       #FB_STATE_TCP_RECONNECTING:
         REGION FB_STATE_TCP_RECONNECTING
           IF #tempTsendcStatus = #TSENDC_EST_OK THEN
             #statErrorAutoCleared := FALSE;
             // Update edge detection
             #statPublishOld := #tempPublish;
             #statSubscribeOld := #tempSubscribe;
             #statUnsubscribeOld := #tempUnsubscribe;
             //Monitor Connection
             #statFBState := #FB_STATE_OPERATING_MONITOR_TCP;
             // Begin MQTT Connection
             #statMqttConnectState := #MQTT_CONNECT_STATE_BUILD_PAKET;
           END_IF;
         END_REGION FB_STATE_TCP_RECONNECTING
       #FB_STATE_DISABLING: // Disabling active
         REGION DISABLING FB
           //  Disabling, e.g. closing connections, etc.
           // When disabling is complete the bit #statDisablingCompleted must be set
           // When MQTT is connected, send disconnect
           IF #statMqttConnectState = #MQTT_CONNECT_STATE_CONNECTED THEN
             IF #statTsendcReq = TRUE THEN
               //Interrupt any existing send jobs
               #statTsendcReq := FALSE;
             ELSE
               // INIT
               #statSendBufferPos := 0;
               //Build fixed Header
               //Message Type
               #statSendBuffer[#statSendBufferPos] := #MQTT_MSG_TYPE_DISCONNECT;
               #statSendBufferPos += 1;
               //Remaining Length (must be O)
               #statSendBuffer[#statSendBufferPos] := #REMAINIG_LEN_0;
               #statSendBufferPos += 1;
               //send request
               #statTsendcLen := #statSendBufferPos;
               #statTsendcReq := TRUE;
               #statMqttConnectState := #MQTT_CONNECT_STATE_DISCONNECTED;
             END_IF;
           ELSE
             //Disable TCP Connection
             #statTsendcReq := FALSE;
             #statTsendcEnable := FALSE;
             #statEnableTimerCommandWatchdog := TRUE;
           END_IF;
           // When TCP connection is closed
           IF #tempTsendcStatus = #TSENDC_DISCONNECTED THEN
             #statEnableTimerCommandWatchdog := FALSE;
             #statDisablingCompleted := TRUE;
           ELSIF #instTimerCommandWatchdog.Q THEN
             #statEnableTimerCommandWatchdog := FALSE;
             #statDisablingCompleted := TRUE;
           END_IF;
         END_REGION DISABLING FB
       ELSE // Undefined state in state machine reached
         #statStatus := #ERR_UNDEFINED_STATE;
         #statErrorUserCleared := TRUE;
     END_CASE;
   END_REGION STATE_MACHINE

   REGION OUTPUTS
     // Write outputs
     IF (#statDisablingCompleted = TRUE) THEN
       // Reset outputs if disabling completed
       #statValid := FALSE;
       #statBusy := FALSE;
       #statError := FALSE;
       #statDone := FALSE;
       #statErrorUserCleared := FALSE;
       #statErrorAutoCleared := FALSE;
       #statStatus := #STATUS_NO_CALL;
       // Reset application specific outputs
       #statRcvMsgStatus := #MSG_DECODE_STATUS_NO_NEW_MSG;
       #statRcvMsgDataLen := 0;

     ELSIF (#statErrorUserCleared = TRUE) AND (#statError = FALSE) THEN
       // Error can only be cleared by user; rising edge at enable input is needed to continue 
       #statValid := FALSE;
       #statBusy := FALSE;
       #statDone := FALSE;
       #statError := TRUE;
       // Write diagnostics
       #diagnostics.status := #statStatus;
       #diagnostics.subfunctionStatus := #statSubfunctionStatus;
       #diagnostics.stateNumber := #statFBErrorState;
       // execution aborted --> set state no processing
       #statTsendcEnable := FALSE; // Terminate Connection, no reason keep it up.
       #statFBState := #FB_STATE_NO_PROCESSING;
       #statMqttConnectState := #MQTT_CONNECT_STATE_NO_PROCESSING;
       #statMqttCommandState := #MQTT_COMMAND_STATE_NO_PROCESSING;
       #statRcvMsgDecodeState := #MSG_DECODE_STATE_NO_PROCESSING;

     ELSIF (#statErrorAutoCleared = TRUE) AND (#statError = FALSE) THEN
       // Error can be reset by FB automatically
       #statValid := FALSE;
       #statBusy := TRUE;
       #statError := TRUE;
       #statDone := FALSE;

       // Write diagnostics
       #diagnostics.status := #statStatus;
       #diagnostics.subfunctionStatus := #statSubfunctionStatus;
       #diagnostics.stateNumber := #statFBErrorState;
       // Handling of autocleared error
       CASE #statStatus OF
           //Just signal error and reset autocleared error afterwards.
         #ERR_MQTT_PAKET_ID_INVALID, #ERR_MQTT_SUBACK_FAILURE, #ERR_MQTT_CONNECT_TIMEOUT,
         #ERR_MQTT_COMMAND_SEND_TIMEOUT, #ERR_MQTT_COMMAND_MULTIPLE_INPUT, #ERR_CNT_EXCEEDS_ARRAY_DIMENSION,
         #ERR_MQTT_COMMAND_PUBLISH_TOPIC_INVALID, #ERR_QOS_INVALID, #ERR_MQTT_COMMAND_SUBSCRIBE_TOPIC_INVALID:
           #statErrorAutoCleared := FALSE;

         ELSE  // Statement section ELSE
           ;
       END_CASE;

     ELSIF (#statErrorAutoCleared = FALSE) AND (#statErrorUserCleared = FALSE) AND (#statError = TRUE) THEN
       // If autocleared error is acknowledged
       #statValid := TRUE;
       #statBusy := TRUE;
       #statError := FALSE;
       #statDone := FALSE;

       //   this line  more detailed status information is used instead of "#STATUS_SUBSEQUENT_CALL"
       CASE #statStatus OF
         #ERR_TCP_RECONNECTING, #ERR_MQTT_CONNECT_TIMEOUT:  // Reconnecting ok, start Mqtt reconnnect
           //set status
           #statStatus := #STATUS_MQTT_CONNECTING;
           //in the following status codes status stays connected. 
         #ERR_MQTT_PAKET_ID_INVALID, #ERR_MQTT_SUBACK_FAILURE, #ERR_MQTT_COMMAND_SEND_TIMEOUT,
         #ERR_MQTT_COMMAND_MULTIPLE_INPUT, #ERR_CNT_EXCEEDS_ARRAY_DIMENSION, #ERR_MQTT_COMMAND_PUBLISH_TOPIC_INVALID,
         #ERR_QOS_INVALID, #ERR_MQTT_COMMAND_SUBSCRIBE_TOPIC_INVALID:
           #statStatus := #STATUS_MQTT_CONNECTED;
         ELSE  // Statement section ELSE
           ;
       END_CASE;
     END_IF;

     // Write static values to outputs
     #valid := #statValid;
     #busy := #statBusy;
     #error := #statError;
     #status := #statStatus;
     //block sets ENO automatically:
     //ENO := TRUE;
     //Write application specific static values to outputs
     #done := #statDone;
     #receivedMsgStatus := #statRcvMsgStatus;
     #receivedMsgDataLen := #statRcvMsgDataLen;
   END_REGION OUTPUTS
END_FUNCTION_BLOCK

FUNCTION "TransmitMqttData" : Void   // FC17, SCL
{ S7_Optimized_Access := 'TRUE' }
VERSION : 0.1
BEGIN
END_FUNCTION

// folder: LMQTT/Utilities

FUNCTION "LMQTT_ConvertToUtf8" : Void   // FC15, SCL
TITLE = LMQTT_ConvertToUtf8
{ S7_Optimized_Access := 'TRUE' }
AUTHOR : SIEMENS
FAMILY : LMQTT
VERSION : 1.0
// Function to convert a WCHAR to a UTF-8 conformant byte sequence
   VAR_INPUT
      character : WChar;   // Character that shall be converted to UTF-8
   END_VAR
   VAR_OUTPUT
      convertedUtf8 : DWord;   // UTF-8 conformant byte sequence. B0 stores first Byte, B1 second and B2 third Byte. B3 is not used
      bytesUsed : USInt;   // Amount of Bytes converted. Ranges from 1 to 3.
      error : Bool;   // TRUE: An error occurred during the execution of the FC
      status : Word;   // 16#0000 - 16#7FFF: Status of the FC, 16#8000 - 16#FFFF: Error identification
   END_VAR
   VAR_TEMP
      tempStatus : Word;   // temp value for output 'status'
      tempConvertedUtf8 : DWord;   // temp value for output 'convertedUtf8'
      tempBytesUsed : USInt;   // temp value for output 'bytesUsed'
      tempCharacter : WChar;   // temp value for input 'character'
   END_VAR
   // Ret_Val : No return for this FC - see error and status output
   VAR CONSTANT
      STATUS_NO_ERROR : Word := 16#0000;   // no error status
      STATUS_EXECUTION_FINISHED : Word := 16#0000;   // Execution finished without errors
      ERR_UNDEFINED : Word := 16#8000;   // Error due to an undefined case
      USINT_NULL : USInt := 0;   // Init value with 0
      DWORD_NULL : DWord := 16#0000_0000;   // Init value with 0
      EMPTY_WCHAR : WChar := WCHAR#' ';   // Empty WChar for comparison
      BELOW_7F : Word := 16#007F;   // Upper limit for character if only one Byte used
      BELOW_7FF : Word := 16#07FF;   // Upper limit for character if two Byte used
      BELOW_MAX_FFFF : Word := 16#FFFF;   // Upper limit for character if three Byte used
      BYTE_3F : Byte := 16#3F;   // Conversion Value
      BYTE_80 : Byte := 16#80;   // Conversion Value
      BYTE_C0 : Byte := 16#C0;   // Conversion Value
      BYTE_E0 : Byte := 16#E0;   // Conversion Value
      USINT_ONE : USInt := 1;   // Const Value to assign amount of bytes used
      USINT_TWO : USInt := 2;   // Const Value to assign amount of bytes used
      USINT_THREE : USInt := 3;   // Const Value to assign amount of bytes used
   END_VAR
BEGIN
   REGION BLOCK INFO HEADER
       //=============================================================================
       // SIEMENS AG
       // (c)Copyright 2020
       //-----------------------------------------------------------------------------
       // Library:       LMQTT
       // Tested with:   CPU 1516-3 PN/DP V2.8
       // Engineering:   TIA Portal V16
       // Restrictions:  --
       // Requirements:  --
       // Functionality: Converts a single WChar Character to a valid UTF-8 encoded byte sequence and saves this to a DWord.
       //                The amount of bytes saved is stored in bytesUsed Output.
       //-----------------------------------------------------------------------------
       // Change log table:
       // Version    Date         Expert in charge         Changes applied
       // 03.00.00   01.10.2020   Siemens Online Support   First released version
       //=============================================================================
   END_REGION

   REGION INITIALISATION  
       // Initialize functionality: reset of variables, diagnostics, etc.
       #tempConvertedUtf8 := #DWORD_NULL;
       #tempBytesUsed := #USINT_NULL;
       #tempStatus := #STATUS_NO_ERROR;
       //assign temp value from input:
        #tempCharacter := #character;

   END_REGION

   REGION PROGRAM LOGIC
       // Use this region for application specific code
       IF #tempCharacter = #EMPTY_WCHAR THEN
           //will be only 1 byte occupied
           #tempConvertedUtf8 := WCHAR_TO_DWORD(#tempCharacter);
           #tempBytesUsed := #USINT_ONE;
       ELSIF (WCHAR_TO_WORD(#tempCharacter) <= (#BELOW_7F)) THEN
           //will be only 1 byte occupied
           #tempConvertedUtf8 := WCHAR_TO_DWORD(#tempCharacter);
           #tempBytesUsed := #USINT_ONE;
       ELSIF (WCHAR_TO_WORD(#tempCharacter) <= (#BELOW_7FF)) THEN
           //will be 2 byte occupied
           #tempConvertedUtf8.%B1 := (WCHAR_TO_BYTE(#tempCharacter) AND #BYTE_3F) OR #BYTE_80;
           #tempConvertedUtf8.%B0 := WORD_TO_BYTE(SHR(IN := WCHAR_TO_WORD(#tempCharacter), N := 6)) OR #BYTE_C0;
           #tempBytesUsed := #USINT_TWO;
       ELSIF (WCHAR_TO_WORD(#tempCharacter) <= (#BELOW_MAX_FFFF)) THEN
           //will be 3 byte occupied
           #tempConvertedUtf8.%B2 := (WCHAR_TO_BYTE(#tempCharacter) AND #BYTE_3F) OR #BYTE_80;
           #tempConvertedUtf8.%B1 := (WORD_TO_BYTE(SHR(IN := WCHAR_TO_WORD(#tempCharacter), N := 6)) AND #BYTE_3F) OR #BYTE_80;
           #tempConvertedUtf8.%B0 := WORD_TO_BYTE(SHR(IN := WCHAR_TO_WORD(#tempCharacter), N := 12)) OR #BYTE_E0;
           #tempBytesUsed := #USINT_THREE;
       END_IF;
   END_REGION

   REGION OUTPUTS
       // Write application specific temp values to outputs
       #bytesUsed := #tempBytesUsed;
       #convertedUtf8 := #tempConvertedUtf8;
       // Write error and status
       #error := #tempStatus.%X15;
       #status := #tempStatus;
       // ENO mechanism is not used --> ENO := TRUE;
       ENO := TRUE;
   END_REGION
END_FUNCTION

// folder: LossManagement

FUNCTION "CopyLoss" : Void   // FC12, SCL
{ S7_Optimized_Access := 'TRUE' }
VERSION : 0.1
   VAR_INPUT
      In : "MachineEventDatatype";
   END_VAR
   VAR_OUTPUT
      Out : "MachineEventListView";
   END_VAR
BEGIN
   #Out."no." := #In.id;
   #Out.LossCode := #In.losscode;
   //#Out.assign_losscode := #In.assign_losscode;
   #Out.Description := "SettingsDB_LossDescription".loss_descriptions[#In.losscode].description;//#In.description;
   //#Out.StartTime:= #In.StartTime;
   //#Out.StartTimeAsStr:= #In.StartTimeAsStr;
   //#Out.EndTime:= #In.EndTime;

   "DTL_to_String"("DTL" := #In.startTime,
                   OutputStr => #Out.StartDateAsStr);


   "DTL_to_String"("DTL" := #In.endTime,
                   OutputStr => #Out.EndDateAsStr);

   "TimeToString"(timeValue := UDINT_TO_TIME(#In.duration),
                  OutputStr => #Out.DurationAsStr);
   //#Out.EndTimeAsStr:= #In.EndTimeAsStr;
   //#Out.DurationAsStr:= #In.DurationAsStr;
   //#Out.Duration := #In.Duration;
   #Out.StatusServer := #In.statusServer;
END_FUNCTION

FUNCTION "CheckDiffLoss" : Void   // FC13, SCL
{ S7_Optimized_Access := 'TRUE' }
VERSION : 0.1
   VAR_INPUT
      "IN 1" : "MachineEventDatatype";
      "IN 2" : "MachineEventListView";
   END_VAR
   VAR_OUTPUT
      IsDiff : Bool;
   END_VAR
BEGIN
   #IsDiff := #"IN 1".id <> #"IN 2"."no.";
   #IsDiff := #IsDiff OR (#"IN 1".losscode <> #"IN 2".LossCode);

   //#IsDiff := #IsDiff OR (#"IN 1".description <> #"IN 2".description);
   // #IsDiff := #IsDiff OR (#"IN 1".StartTimeAsStr <> #"IN 2".StartTimeAsStr);
   // #IsDiff := #IsDiff OR (#"IN 1".EndTimeAsStr <> #"IN 2".EndTimeAsStr);
   // #IsDiff := #IsDiff OR (#"IN 1".DurationAsStr <> #"IN 2".DurationAsStr);
   #IsDiff := #IsDiff OR (#"IN 1".statusServer <> #"IN 2".StatusServer);
END_FUNCTION

FUNCTION "ListviewDisplayLoss" : Void   // FC14, SCL
{ S7_Optimized_Access := 'TRUE' }
VERSION : 0.1
   VAR_INPUT
      MinSlotId : Int;
      MaxSlotId : Int;
   END_VAR
   VAR_TEMP
      tmpIsDiff : Bool;
   END_VAR
BEGIN
   // FOR "bufferLossId" := 1 TO 30 DO
   //     IF "BuffersLoss_DB".buffer_loss_in_shift["bufferLossId"].id > 0 THEN

   //         IF ("slotId" > #MinSlotId) AND ("slotId" <= #MaxSlotId) THEN
   //             IF "listviewId" <= 10 THEN

   //                 // "CheckDiffLoss"("IN 1" := "BuffersLoss_DB".buffer_loss_in_shift["bufferLossId"],
   //                 //                 "IN 2" := "DB_Machine".machine_event_listview["listviewId"],
   //                 //                 IsDiff => #tmpIsDiff);
   //                 #tmpIsDiff := TRUE;
   //                 IF #tmpIsDiff THEN
   //                     "CopyLoss"(In := "BuffersLoss_DB".buffer_loss_in_shift["bufferLossId"],
   //                                Out => "DB_Machine".machine_event_listview["listviewId"]);
   //                 END_IF;
   //                 //
   //                 "DB_Machine".machine_event_listview["listviewId"].IsHaveData := TRUE;
   //                 "listviewId" := "listviewId" + 1;
   //             END_IF;
   //             //
   //         END_IF;

   //         "slotId" := "slotId" + 1;
   //     END_IF;
   // END_FOR;
END_FUNCTION

FUNCTION "ShowDescriptionLossByGroupId" : Void   // FC22, SCL
{ S7_Optimized_Access := 'TRUE' }
VERSION : 0.1
   VAR_INPUT
      GroupId : USInt;
      PageCurrent : UDInt;
      NumberDataEachPage : USInt;
   END_VAR
   VAR_OUTPUT
      ListDescriptionResult : Array[1..10] of String[30];
   END_VAR
   VAR_TEMP
      IndexFor : USInt;
      ListDescriptionResultTemp : Array[1..100] of String[30];
      IndexLossResult : USInt;
   END_VAR
BEGIN
   IF #GroupId>=1 AND #GroupId<=10 THEN
       #IndexLossResult := 1;
       FOR #IndexFor := 1 TO 100 DO
           IF "SettingsDB_LossDescription".loss_descriptions[#IndexFor].group_id = #GroupId THEN // Statement section FOR
               #ListDescriptionResultTemp[#IndexLossResult] := "SettingsDB_LossDescription".loss_descriptions[#IndexFor].description;
               #IndexLossResult += 1;
           END_IF;
       END_FOR;

       FOR #IndexFor := 1 TO 10 DO
           IF #IndexLossResult <= 10 THEN
               #ListDescriptionResult[#IndexLossResult] := '';
               //#ListDescriptionResult[#IndexLossResult].group_id := 0;
               #IndexLossResult += 1;
           ELSE
               EXIT;
           END_IF;
       END_FOR;

   ELSIF #GroupId=0 THEN //Case All
       FOR #IndexFor := 1 TO 10 DO
           #ListDescriptionResult[#IndexFor] := "SettingsDB_LossDescription".loss_descriptions[#IndexFor + (#PageCurrent - 1) * #NumberDataEachPage].description;
       END_FOR;
   END_IF;
END_FUNCTION

FUNCTION "MappingLossGroup" : Void   // FC23, SCL
{ S7_Optimized_Access := 'TRUE' }
VERSION : 0.1
   VAR_TEMP
      indexFor : USInt;
   END_VAR
BEGIN
   FOR #indexFor := 1 TO 10 DO
       IF "SettingsDB_LossDescription".loss_name_group[#indexFor] = '' THEN
           "DB_DataHMI".VisibleCheckboxLossGroup[#indexFor] := FALSE;
       ELSE
           "DB_DataHMI".VisibleCheckboxLossGroup[#indexFor] := TRUE;
       END_IF;

       "DB_DataHMI".LossGroupHmiDTO[#indexFor] := "SettingsDB_LossDescription".loss_name_group[#indexFor];
   END_FOR;
END_FUNCTION

FUNCTION "GetBufferHistoricalShowHMI" : Void   // FC24, SCL
{ S7_Optimized_Access := 'TRUE' }
VERSION : 0.1
   VAR_INPUT
      page_current_hmi : UDInt;
   END_VAR
   VAR_TEMP
      index_for : USInt;
      index_buffer : UDInt;
      page_hmi_cvt : UDInt;
   END_VAR
BEGIN
   IF #page_current_hmi>=1 THEN
       #page_hmi_cvt := #page_current_hmi MOD 10;
       IF #page_hmi_cvt=0 THEN
           #page_hmi_cvt := 10;
       END_IF;

       #index_buffer := (#page_hmi_cvt - 1) * 5;

       FOR #index_for:= 1 TO 5 DO
           IF "BuffersLoss_DB".buffer_loss_in_historical[#index_buffer + #index_for].id > 0 THEN
               "DB_DataHMI".DataLossHistoricalShowHmiDTO[#index_for]."no." := UDINT_TO_UINT((#page_current_hmi - 1) * 5 + #index_for);
               "DB_DataHMI".DataLossHistoricalShowHmiDTO[#index_for].LossCode := "BuffersLoss_DB".buffer_loss_in_historical[#index_buffer + #index_for].losscode;

               "Cvt_Duration_to_String"("Time(ms)" := "BuffersLoss_DB".buffer_loss_in_historical[#index_buffer + #index_for].duration,
                                        ConvertTimeToStr => "DB_DataHMI".DataLossHistoricalShowHmiDTO[#index_for].DurationAsStr);

               "DTL_to_DateString"("DTL" := "BuffersLoss_DB".buffer_loss_in_historical[#index_buffer + #index_for].startTime,
                                   DateTimeString => "DB_DataHMI".DataLossHistoricalShowHmiDTO[#index_for].StartDateAsStr);
               "DTL_to_TimeString"("DTL" := "BuffersLoss_DB".buffer_loss_in_historical[#index_buffer + #index_for].startTime,
                                   DateTimeString => "DB_DataHMI".DataLossHistoricalShowHmiDTO[#index_for].StartTimeAsStr);

               "DTL_to_DateString"("DTL" := "BuffersLoss_DB".buffer_loss_in_historical[#index_buffer + #index_for].endTime,
                                   DateTimeString => "DB_DataHMI".DataLossHistoricalShowHmiDTO[#index_for].EndDateAsStr);
               "DTL_to_TimeString"("DTL" := "BuffersLoss_DB".buffer_loss_in_historical[#index_buffer + #index_for].endTime,
                                   DateTimeString => "DB_DataHMI".DataLossHistoricalShowHmiDTO[#index_for].EndTimeAsStr);

               IF  "DB_DataHMI".DataLossHistoricalShowHmiDTO[#index_for].LossCode>0 AND  "DB_DataHMI".DataLossHistoricalShowHmiDTO[#index_for].LossCode<=100 THEN
                   "DB_DataHMI".DataLossHistoricalShowHmiDTO[#index_for].Description := "SettingsDB_LossDescription".loss_descriptions["DB_DataHMI".DataLossHistoricalShowHmiDTO[#index_for].LossCode].description;
                   IF "SettingsDB_LossDescription".loss_descriptions["DB_DataHMI".DataLossHistoricalShowHmiDTO[#index_for].LossCode].group_id>0 AND
                       "SettingsDB_LossDescription".loss_descriptions["DB_DataHMI".DataLossHistoricalShowHmiDTO[#index_for].LossCode].group_id<=10 THEN
                       "DB_DataHMI".DataLossHistoricalShowHmiDTO[#index_for].GroupLossReason := "SettingsDB_LossDescription".loss_name_group["SettingsDB_LossDescription".loss_descriptions["DB_DataHMI".DataLossHistoricalShowHmiDTO[#index_for].LossCode].group_id];
                   END_IF;
               END_IF;

               "DB_DataHMI".DataLossHistoricalShowHmiDTO[#index_for].IsHaveData := TRUE;
           END_IF;
       END_FOR;
   END_IF;
END_FUNCTION

FUNCTION "LogStartLoss" : Void   // FC26, SCL
{ S7_Optimized_Access := 'TRUE' }
VERSION : 0.1
BEGIN
   "GLobalDB_LossManagementDB".current_status_machine.startTime := "GlobalDB_RTC".RTC_Local;
END_FUNCTION

FUNCTION "LogEndLoss" : Void   // FC27, SCL
{ S7_Optimized_Access := 'TRUE' }
VERSION : 0.1
BEGIN
   "GLobalDB_LossManagementDB".current_status_machine.startTime := "GlobalDB_RTC".RTC_Local;
END_FUNCTION

FUNCTION "CheckMoveDataLossCurrent" : Void   // FC28, SCL
{ S7_Optimized_Access := 'TRUE' }
VERSION : 0.1
BEGIN
   "GLobalDB_LossManagementDB".current_status_machine.endTime := "GlobalDB_RTC".RTC_Local;
   "GLobalDB_LossManagementDB".current_status_machine.duration := "GLobalDB_LossManagementDB"."duration_status_curent(ms)";
   "GLobalDB_LossManagementDB".current_status_machine.id := "GLobalDB_LossManagementDB".id_loss;


   "DTL_to_StringV2"("DTL":="GLobalDB_LossManagementDB".current_status_machine.startTime,
                     DateTimeString=>"DB_DataHMI".PageHomeStartTimeStatusCurrent);

   "DTL_to_StringV2"("DTL" := "GLobalDB_LossManagementDB".current_status_machine.endTime,
                     DateTimeString => "DB_DataHMI".PageHomeEndTimeStatusCurrent);

   "Cvt_Duration_to_String"("Time(ms)":="GLobalDB_LossManagementDB".current_status_machine.duration,
                            ConvertTimeToStr=>"DB_DataHMI".PageHomeDurationStatusCurrent);


   //Kiểm tra Loss hiện tại quá tgian cài đặt sẽ bắt buộc "AssignLoss"
   IF ("GLobalDB_LossManagementDB".current_status_machine.duration/1000) >= ("DataSetting"."TimeThresholdShowWarningAssignLoss(s)")
       AND "DB_DataHMI".FlagCancelAssignLossCurrent=FALSE
       AND ("DB_DataHMI".MachineStatus=2 OR "DB_DataHMI".MachineStatus=3) THEN
       "DB_DataHMI".PageHomeBitShowAssignLoss := TRUE;
       "DB_DataHMI".TypeAssignLoss := 3;
   ELSE
       "DB_DataHMI".PageHomeBitShowAssignLoss := FALSE;
   END_IF;


   //Kiểm tra  AssignLoss hiện tại để move data
   IF "DB_DataHMI".EventAssignLossCurrent=TRUE THEN
       "DB_DataHMI".StartTimeAssignLossCurrent := "DB_DataHMI".PageHomeStartTimeStatusCurrent;
       "DB_DataHMI".EndTimeAssignLossCurrent := "DB_DataHMI".PageHomeEndTimeStatusCurrent;
       "DB_DataHMI".DurationAssignLossCurrent := "DB_DataHMI".PageHomeDurationStatusCurrent;
   END_IF;


   //MOve tamj ddons khacsh
   IF "DB_DataHMI".MachineStatus=2 OR "DB_DataHMI".MachineStatus=3 THEN
       "GLobalDB_LossManagementDB".current_status_machine.statusServer := UINT_TO_USINT("DB_DataHMI".MachineStatus);

       "BuffersLoss_DB".buffer_loss_in_shift["GLobalDB_LossManagementDB".index_buffer_loss_in_shift_current].startTime := "GLobalDB_LossManagementDB".current_status_machine.startTime;
       "BuffersLoss_DB".buffer_loss_in_shift["GLobalDB_LossManagementDB".index_buffer_loss_in_shift_current].endTime := "GlobalDB_RTC".RTC_Defaul;
       "BuffersLoss_DB".buffer_loss_in_shift["GLobalDB_LossManagementDB".index_buffer_loss_in_shift_current].id := "GLobalDB_LossManagementDB".current_status_machine.id;
       "BuffersLoss_DB".buffer_loss_in_shift["GLobalDB_LossManagementDB".index_buffer_loss_in_shift_current].duration := "GLobalDB_LossManagementDB".current_status_machine.duration;
       "BuffersLoss_DB".buffer_loss_in_shift["GLobalDB_LossManagementDB".index_buffer_loss_in_shift_current].statusServer := "GLobalDB_LossManagementDB".current_status_machine.statusServer;
   END_IF;
END_FUNCTION

FUNCTION "LogLoss" : Void   // FC33, SCL
{ S7_Optimized_Access := 'TRUE' }
VERSION : 0.1
   VAR_INPUT
      status : UInt;   // 1: Runnig, 2Stop, 3Idle
   END_VAR
   VAR_IN_OUT
      index_buffer : USInt;   // 1=>100
   END_VAR
BEGIN
   IF #index_buffer>=1 AND #index_buffer<=100 THEN
       "BuffersLoss_DB".buffer_loss_in_shift[#index_buffer] := "GLobalDB_LossManagementDB".current_status_machine;
       "BuffersLoss_DB".buffer_loss_in_shift[#index_buffer].statusServer := UINT_TO_USINT(#status);

       "GLobalDB_LossManagementDB".id_loss += 1;
       //"DB_Machine".NumberLossInShift += 1;
       #index_buffer += 1;
       IF #index_buffer > 100 THEN
           #index_buffer := 1;
       END_IF;
   ELSE
       #index_buffer := 1;
   END_IF;
END_FUNCTION

FUNCTION "CheckIndexRowAssignLoss" : Void   // FC42, SCL
{ S7_Optimized_Access := 'TRUE' }
VERSION : 0.1
   VAR_TEMP
      index_for : USInt;
      group_id : UInt;
   END_VAR
BEGIN
   FOR #index_for := 1 TO 5 DO
       IF "DB_DataHMI".EventIndexRowInShift[#index_for]=TRUE THEN
           "DB_DataHMI".IndexRowAssignLoss := #index_for;
           "DB_DataHMI".EventIndexRowInShift[#index_for] := FALSE;

           "DB_DataHMI".TypeAssignLoss := 1;
       END_IF;
   END_FOR;

   FOR #index_for := 1 TO 5 DO
       IF "DB_DataHMI".EventIndexRowHistorical[#index_for] = TRUE THEN
           "DB_DataHMI".IndexRowAssignLoss := #index_for;
           "DB_DataHMI".EventIndexRowHistorical[#index_for] := FALSE;

           "DB_DataHMI".TypeAssignLoss := 2;
       END_IF;
   END_FOR;



   IF "DB_DataHMI".TypeAssignLoss=1 THEN //LOss In Shift
       "DB_DataHMI".LossReasonSelectId := 0;
       IF "DB_DataHMI".IndexRowAssignLoss>=1 AND "DB_DataHMI".IndexRowAssignLoss<=5 THEN
           "DB_DataHMI".StartTimeAssignLossCurrent := CONCAT(IN1 := "DB_DataHMI".DataLossInShiftShowHmiDTO["DB_DataHMI".IndexRowAssignLoss].StartDateAsStr,
                                                             IN2 := ' ',
                                                             IN3 := "DB_DataHMI".DataLossInShiftShowHmiDTO["DB_DataHMI".IndexRowAssignLoss].StartTimeAsStr);

           "DB_DataHMI".EndTimeAssignLossCurrent := CONCAT(IN1 := "DB_DataHMI".DataLossInShiftShowHmiDTO["DB_DataHMI".IndexRowAssignLoss].EndDateAsStr,
                                                             IN2 := ' ',
                                                             IN3 := "DB_DataHMI".DataLossInShiftShowHmiDTO["DB_DataHMI".IndexRowAssignLoss].EndTimeAsStr);
           "DB_DataHMI".DurationAssignLossCurrent := "DB_DataHMI".DataLossInShiftShowHmiDTO["DB_DataHMI".IndexRowAssignLoss].DurationAsStr;

           //Tim thông tin AssignLoss của Loss hiện tại nếu có
           "ResetCheckBoxLossReason"();
           IF "DB_DataHMI".DataLossInShiftShowHmiDTO["DB_DataHMI".IndexRowAssignLoss].LossCode>0 AND "DB_DataHMI".DataLossInShiftShowHmiDTO["DB_DataHMI".IndexRowAssignLoss].LossCode<=10 THEN
               "DB_DataHMI".CheckboxLossReason["DB_DataHMI".DataLossInShiftShowHmiDTO["DB_DataHMI".IndexRowAssignLoss].LossCode] := 1;

               "DB_DataHMI".LossReasonSelectId := "DB_DataHMI".DataLossInShiftShowHmiDTO["DB_DataHMI".IndexRowAssignLoss].LossCode;

               "ResetCheckBoxLossGroup"();
               #group_id := "SettingsDB_LossDescription".loss_descriptions["DB_DataHMI".DataLossInShiftShowHmiDTO["DB_DataHMI".IndexRowAssignLoss].LossCode].group_id;
               IF #group_id>0 AND #group_id<=10 THEN
                   "DB_DataHMI".CheckboxLossGroup[#group_id] := 1;
               END_IF;

           END_IF;
       END_IF;
       "DB_DataHMI".TypeAssignLoss := 0;
   ELSIF "DB_DataHMI".TypeAssignLoss=2 THEN //Historical
       "DB_DataHMI".LossReasonSelectId := 0;
       IF "DB_DataHMI".IndexRowAssignLoss >= 1 AND "DB_DataHMI".IndexRowAssignLoss <= 5 THEN
           "DB_DataHMI".StartTimeAssignLossCurrent := CONCAT(IN1 := "DB_DataHMI".DataLossHistoricalShowHmiDTO["DB_DataHMI".IndexRowAssignLoss].StartDateAsStr,
                                                             IN2 := ' ',
                                                             IN3 := "DB_DataHMI".DataLossHistoricalShowHmiDTO["DB_DataHMI".IndexRowAssignLoss].EndTimeAsStr);

           "DB_DataHMI".EndTimeAssignLossCurrent := CONCAT(IN1 := "DB_DataHMI".DataLossHistoricalShowHmiDTO["DB_DataHMI".IndexRowAssignLoss].EndDateAsStr,
                                                           IN2 := ' ',
                                                           IN3 := "DB_DataHMI".DataLossHistoricalShowHmiDTO["DB_DataHMI".IndexRowAssignLoss].EndTimeAsStr);
           "DB_DataHMI".DurationAssignLossCurrent := "DB_DataHMI".DataLossHistoricalShowHmiDTO["DB_DataHMI".IndexRowAssignLoss].DurationAsStr;


           //Tim thông tin AssignLoss của Loss hiện tại nếu có
           "ResetCheckBoxLossReason"();
           IF "DB_DataHMI".DataLossHistoricalShowHmiDTO["DB_DataHMI".IndexRowAssignLoss].LossCode > 0 AND
               "DB_DataHMI".DataLossHistoricalShowHmiDTO["DB_DataHMI".IndexRowAssignLoss].LossCode <= 10 THEN
               "DB_DataHMI".CheckboxLossReason["DB_DataHMI".DataLossHistoricalShowHmiDTO["DB_DataHMI".IndexRowAssignLoss].LossCode] := 1;

               "DB_DataHMI".LossReasonSelectId := "DB_DataHMI".DataLossHistoricalShowHmiDTO["DB_DataHMI".IndexRowAssignLoss].LossCode;

               "ResetCheckBoxLossGroup"();
               #group_id := "SettingsDB_LossDescription".loss_descriptions["DB_DataHMI".DataLossHistoricalShowHmiDTO["DB_DataHMI".IndexRowAssignLoss].LossCode].group_id;
               IF #group_id > 0 AND #group_id <= 10 THEN
                   "DB_DataHMI".CheckboxLossGroup[#group_id] := 1;
               END_IF;

           END_IF;
       END_IF;
       "DB_DataHMI".TypeAssignLoss := 0;
   ELSIF "DB_DataHMI".TypeAssignLoss=3 THEN //Loss Current
       "DB_DataHMI".StartTimeAssignLossCurrent := "DB_DataHMI".PageHomeStartTimeStatusCurrent;
       "DB_DataHMI".EndTimeAssignLossCurrent := "DB_DataHMI".PageHomeEndTimeStatusCurrent;
       "DB_DataHMI".DurationAssignLossCurrent := "DB_DataHMI".PageHomeDurationStatusCurrent;
   END_IF;


   //Kiểm tra Action Cancel nếu người ta bỏ qua AssignLoss hiện tại
   IF "DB_DataHMI".FlagCancelAssignLossCurrent = TRUE AND "DB_DataHMI".TypeAssignLoss=3 THEN
       "DB_DataHMI".PageHomeBitShowAssignLoss := FALSE;
   END_IF;
END_FUNCTION

FUNCTION "FindSyncLossInShift" : Void   // FC63, SCL
{ S7_Optimized_Access := 'TRUE' }
VERSION : 0.1
   VAR_TEMP
      index_for : USInt;
      compare_start_time : Bool;
      compare_end_time : Bool;
   END_VAR
BEGIN
   FOR #index_for := 1 TO 100 DO
       "CompareDTL"(DTL_Input1:="DB_Server".LossInShiftAssign.startTime,
                                          DTL_Input2:="BuffersLoss_DB".buffer_loss_in_shift[#index_for].startTime,
                                          Result=>#compare_start_time);

                             "CompareDTL"(DTL_Input1 := "DB_Server".LossInShiftAssign.endTime,
                                           DTL_Input2 := "BuffersLoss_DB".buffer_loss_in_shift[#index_for].endTime,
                                           Result => #compare_end_time);

      IF #compare_start_time = TRUE AND #compare_end_time = TRUE THEN
          "BuffersLoss_DB".buffer_loss_in_shift[#index_for].losscode := "DB_Server".LossInShiftAssign.losscode;
          EXIT;
      END_IF;
   END_FOR;
END_FUNCTION

FUNCTION "ResStatusSearchLossHistorical" : Void   // FC69, SCL
{ S7_Optimized_Access := 'TRUE' }
VERSION : 0.1
   VAR_IN_OUT
      value_flag : UInt;
   END_VAR
BEGIN
   IF #value_flag=2 THEN
       "DB_DataHMI".EventBitShowPopupLoading := FALSE;
       IF "DB_Server".PageHistorical.TotalData=0 THEN
           "DB_DataHMI".EventBitShowNoDataHistorical := TRUE;
           "DB_Server".ActionSearchLossHistorical := 3;
       END_IF;
   ELSIF #value_flag=4 THEN
       "DB_DataHMI".EventBitShowPopupLoading := FALSE;
       "DB_DataHMI".EventBitShowPopupErrorFormatDaySearch := TRUE;
       #value_flag := 3;
   END_IF;
END_FUNCTION

// folder: RTC

FUNCTION "RTC" : Void   // FC6, LAD
{ S7_Optimized_Access := 'TRUE' }
VERSION : 0.1
   VAR_OUTPUT
      Year : UInt;
      Month : UInt;
      Day : UInt;
      Hour : UInt;
      Minute : UInt;
      Second : UInt;
   END_VAR
   VAR_TEMP
      max : USInt;
      min : USInt;
   END_VAR
BEGIN

REGION Network 1
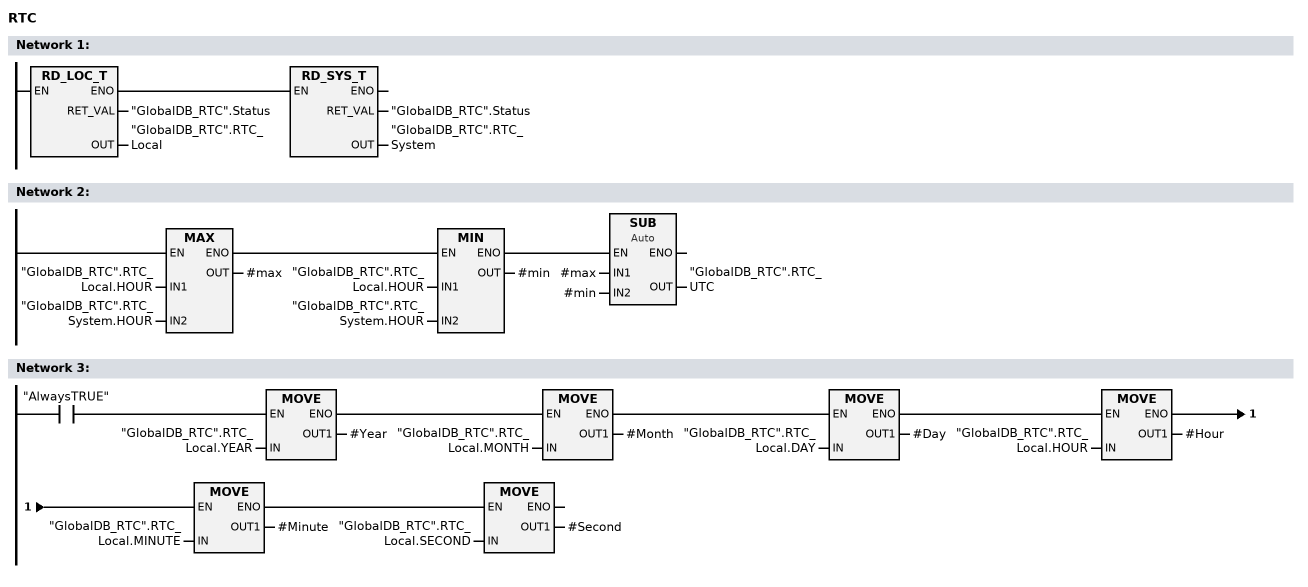
   // ENO of a box is taken as its EN; it also drops when the box reports an error
   "GlobalDB_RTC".Status := RD_LOC_T(OUT => "GlobalDB_RTC".RTC_Local);
   "GlobalDB_RTC".Status := RD_SYS_T(OUT => "GlobalDB_RTC".RTC_System);
END_REGION

REGION Network 2
   #max := MAX(IN1 := "GlobalDB_RTC".RTC_Local.HOUR, IN2 := "GlobalDB_RTC".RTC_System.HOUR);
   #min := MIN(IN1 := "GlobalDB_RTC".RTC_Local.HOUR, IN2 := "GlobalDB_RTC".RTC_System.HOUR);
   "GlobalDB_RTC".RTC_UTC := #max - #min;
END_REGION

REGION Network 3
   RUNG wire#powerrail
      Contact( "AlwaysTRUE" )
      Move(in := "GlobalDB_RTC".RTC_Local.YEAR, out1 => #Year)
      Move(in := "GlobalDB_RTC".RTC_Local.MONTH, out1 => #Month)
      Move(in := "GlobalDB_RTC".RTC_Local.DAY, out1 => #Day)
      Move(in := "GlobalDB_RTC".RTC_Local.HOUR, out1 => #Hour)
      Move(in := "GlobalDB_RTC".RTC_Local.MINUTE, out1 => #Minute)
      Move(in := "GlobalDB_RTC".RTC_Local.SECOND, out1 => #Second)
   END_RUNG
   // the same network as SCL:
   IF "AlwaysTRUE" THEN
       #Year := "GlobalDB_RTC".RTC_Local.YEAR;
       #Month := "GlobalDB_RTC".RTC_Local.MONTH;
       #Day := "GlobalDB_RTC".RTC_Local.DAY;
       #Hour := "GlobalDB_RTC".RTC_Local.HOUR;
       #Minute := "GlobalDB_RTC".RTC_Local.MINUTE;
       #Second := "GlobalDB_RTC".RTC_Local.SECOND;
   END_IF;
END_REGION
END_FUNCTION

FUNCTION "SyncTimeFromPC" : Void   // FC66, LAD
{ S7_Optimized_Access := 'TRUE' }
VERSION : 0.1
   VAR_IN_OUT
      EventSync : Bool;
   END_VAR
BEGIN

REGION Network 1: Set và Get lại thời gian PLC khi có sự kiện update
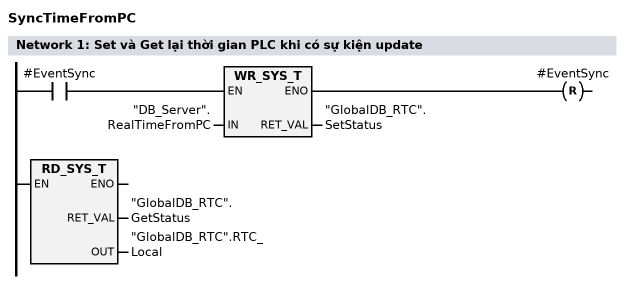
   // ENO of a box is taken as its EN; it also drops when the box reports an error
   IF #EventSync THEN
       "GlobalDB_RTC".SetStatus := WR_SYS_T(IN := "DB_Server".RealTimeFromPC);
       #EventSync := FALSE;
   END_IF;
   "GlobalDB_RTC".GetStatus := RD_SYS_T(OUT => "GlobalDB_RTC".RTC_Local);
END_REGION
END_FUNCTION

// folder: Sensor-Counter

FUNCTION_BLOCK "CounterFB"   // FB3, LAD
{ S7_Optimized_Access := 'TRUE' }
VERSION : 0.1
   VAR_INPUT
      bCounterTrigger : Bool;
      bResetCounter : Bool;
      TonFilter_x1ms : UInt := 10;   // ms
      ToffFilter_x1ms : UInt := 10;   // ms
   END_VAR
   VAR_IN_OUT
      CounterOut : UDInt;
   END_VAR
   VAR RETAIN
      P_tmp : Bool;
      N_tmp : Bool;
   END_VAR
   VAR
      Ton_start : Bool;
      Toff_start : Bool;
   END_VAR
   VAR RETAIN
      IEC_Ton : IEC_TIMER;
      IEC_Toff : IEC_TIMER;
      bTmp : Bool;
   END_VAR
   VAR
      Ton_x1ms : Time;
      Toff_x1ms : Time;
   END_VAR
   VAR_TEMP   // added for the SCL form of the ladder/FBD networks
      _w1 : Bool;
   END_VAR
BEGIN

REGION Network 1
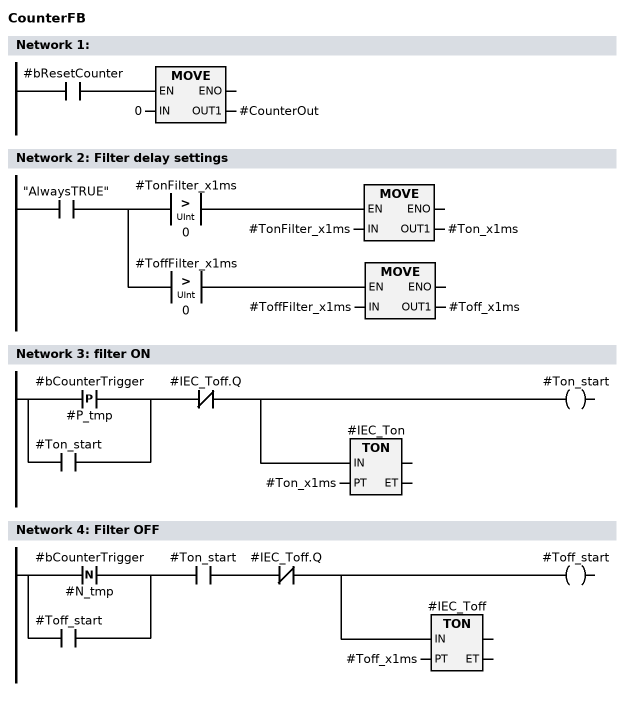
   RUNG wire#powerrail
      Contact( #bResetCounter )
      Move(in := 0, out1 => #CounterOut)
   END_RUNG
   // the same network as SCL:
   IF #bResetCounter THEN #CounterOut := 0; END_IF;
END_REGION

REGION Network 2: Filter delay settings
   RUNG wire#powerrail
      Contact( "AlwaysTRUE" )
      wire#w1
      { S7_Templates := "SrcType := UInt" } GT_Contact(in1 := #TonFilter_x1ms, in2 := 0)
      Move(in := #TonFilter_x1ms, out1 => #Ton_x1ms)
   END_RUNG
   RUNG wire#w1
      { S7_Templates := "SrcType := UInt" } GT_Contact(in1 := #ToffFilter_x1ms, in2 := 0)
      Move(in := #ToffFilter_x1ms, out1 => #Toff_x1ms)
   END_RUNG
   // the same network as SCL:
   IF "AlwaysTRUE" AND (#TonFilter_x1ms > 0) THEN #Ton_x1ms := #TonFilter_x1ms; END_IF;
   IF "AlwaysTRUE" AND (#ToffFilter_x1ms > 0) THEN #Toff_x1ms := #ToffFilter_x1ms; END_IF;
END_REGION

REGION Network 3: filter ON
   #_w1 := #bCounterTrigger AND NOT #P_tmp;   // rising edge of #bCounterTrigger
   #P_tmp := #bCounterTrigger;
   #Ton_start := (#_w1 OR #Ton_start) AND NOT #IEC_Toff.Q;
   #IEC_Ton.TON(IN := #Ton_start, PT := #Ton_x1ms);
END_REGION

REGION Network 4: Filter OFF
   #_w1 := NOT #bCounterTrigger AND #N_tmp;   // falling edge of #bCounterTrigger
   #N_tmp := #bCounterTrigger;
   #Toff_start := (#_w1 OR #Toff_start) AND #Ton_start AND NOT #IEC_Toff.Q;
   #IEC_Toff.TON(IN := #Toff_start, PT := #Toff_x1ms);
END_REGION

REGION Network 5 (SCL)
   IF #Ton_start AND NOT #bTmp THEN
       #CounterOut := #CounterOut + 1;
   END_IF;
   #bTmp := #Ton_start;
END_REGION
END_FUNCTION_BLOCK

// folder: Sensor-Speed

FUNCTION_BLOCK "1.2 Speed_Sensor"   // FB1, LAD
{ S7_Optimized_Access := 'TRUE' }
VERSION : 0.1
   VAR_INPUT
      "InputTimeSpeed(time_each_pulse)" : Time;
      NumberOfGears : UInt;
      Index : Int;
   END_VAR
   VAR_OUTPUT
      "OutputSpeed(rpm)" : DInt;
      "TimePerPulse(x1ms)" : DInt;
   END_VAR
   VAR RETAIN
      bThroudoutStart : Bool;
      TimeSpeed : Time;
      speed_tmp : Array[1..3] of DInt;
      speed_tmpidx : Int;
      previous_speed_tmpidx : Int;
      CurrentSpeed : DInt;
   END_VAR
   VAR
      real_tmp : Real;
      real_tmp_1 : Real;
      dint_tmp : DInt;
      real_tmp_2 : Real;
      number_of_gears_tmp : Real;
   END_VAR
   VAR_TEMP   // added for the SCL form of the ladder/FBD networks
      _w1 : Bool;
   END_VAR
BEGIN

REGION Network 1
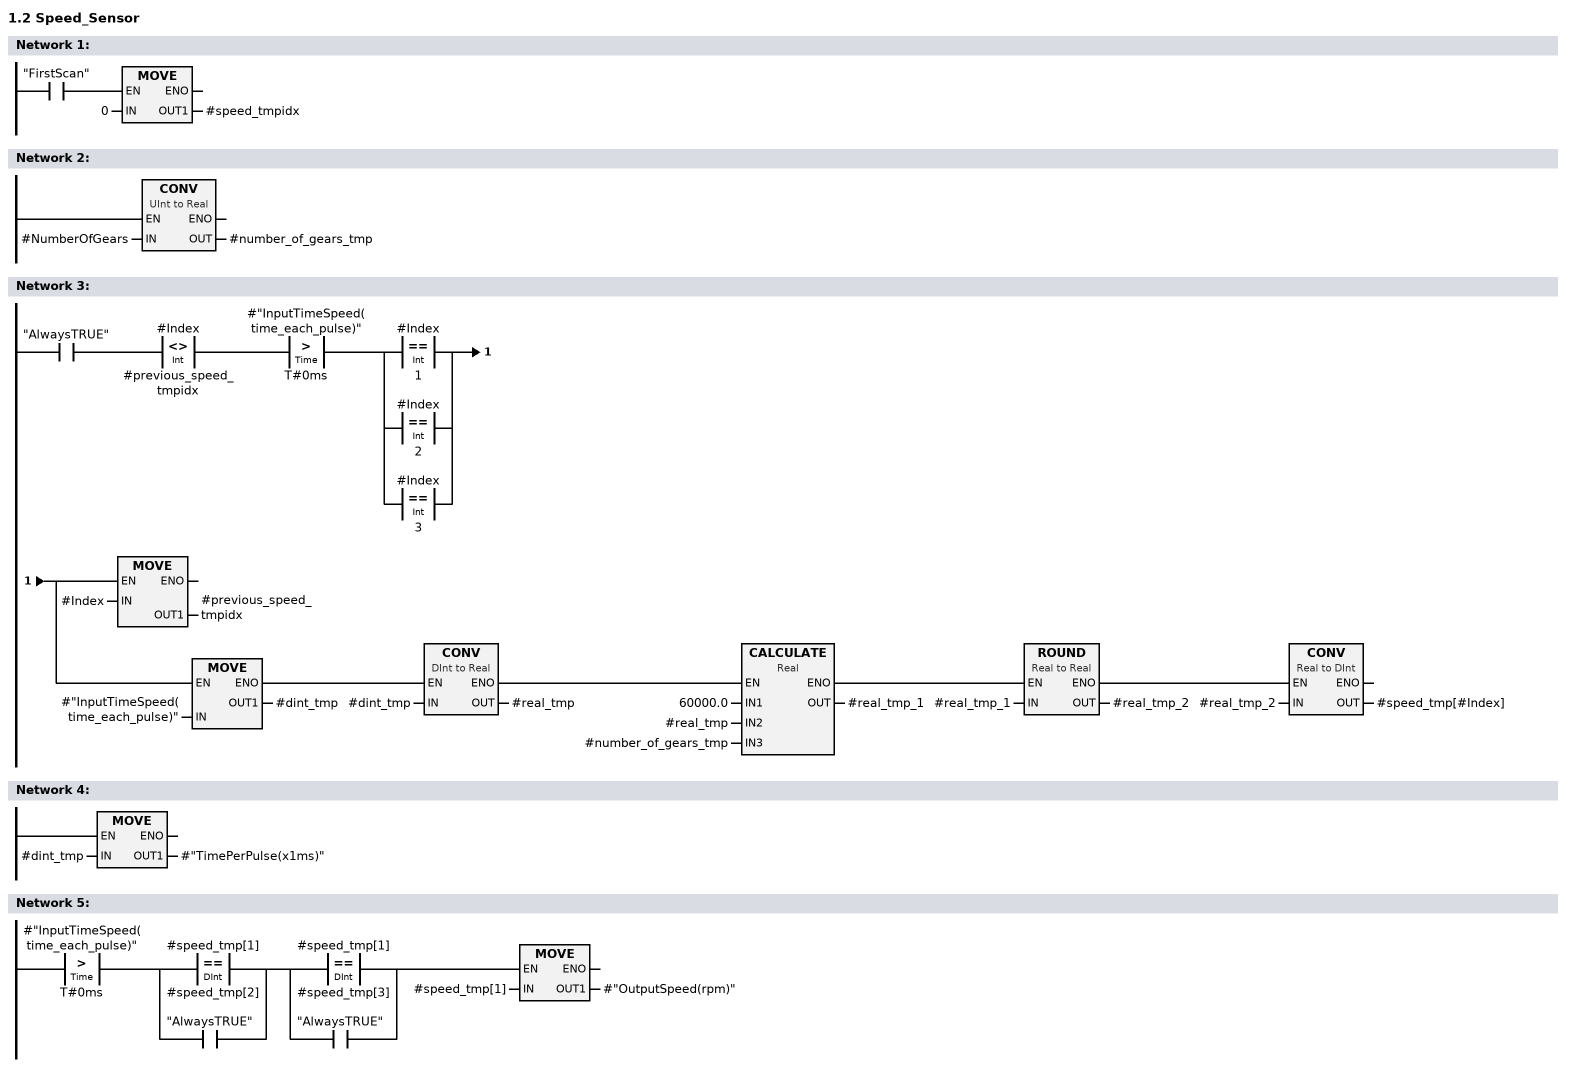
   RUNG wire#powerrail
      Contact( "FirstScan" )
      Move(in := 0, out1 => #speed_tmpidx)
   END_RUNG
   // the same network as SCL:
   IF "FirstScan" THEN #speed_tmpidx := 0; END_IF;
END_REGION

REGION Network 2
   RUNG wire#powerrail
      { S7_Templates := "[SrcType := UInt, DestType := Real]" } Convert(in := #NumberOfGears, out => #number_of_gears_tmp)
   END_RUNG
   // the same network as SCL:
   #number_of_gears_tmp := UINT_TO_REAL(#NumberOfGears);
END_REGION

REGION Network 3
   RUNG wire#powerrail
      Contact( "AlwaysTRUE" )
      { S7_Templates := "SrcType := Int" } NE_Contact(in1 := #Index, in2 := #previous_speed_tmpidx)
      { S7_Templates := "SrcType := Time" } GT_Contact(in1 := #"InputTimeSpeed(time_each_pulse)", in2 := T#0ms)
      wire#w1
      { S7_Templates := "SrcType := Int" } EQ_Contact(in1 := #Index, in2 := 1)
      wire#w2
      Move(in := #Index, out1 => #previous_speed_tmpidx)
   END_RUNG
   RUNG wire#w1
      { S7_Templates := "SrcType := Int" } EQ_Contact(in1 := #Index, in2 := 2)
   END_RUNG wire#w2
   RUNG wire#w1
      { S7_Templates := "SrcType := Int" } EQ_Contact(in1 := #Index, in2 := 3)
   END_RUNG wire#w2
   RUNG wire#w2
      Move(in := #"InputTimeSpeed(time_each_pulse)", out1 => #dint_tmp)
      { S7_Templates := "[SrcType := DInt, DestType := Real]" } Convert(in := #dint_tmp, out => #real_tmp)
      { S7_Templates := "SrcType := Real"; S7_Expression := "IN1/(IN2*IN3)" } Calculate(in1 := 60000.0, in2 := #real_tmp, in3 := #number_of_gears_tmp, out => #real_tmp_1)
      { S7_Templates := "[SrcType := Real, DestType := Real]" } Round(in := #real_tmp_1, out => #real_tmp_2)
      { S7_Templates := "[SrcType := Real, DestType := DInt]" } Convert(in := #real_tmp_2, out => #speed_tmp[#Index])
   END_RUNG
   // the same network as SCL:
   #_w1 := "AlwaysTRUE" AND (#Index <> #previous_speed_tmpidx) AND (#"InputTimeSpeed(time_each_pulse)" > T#0ms) AND ((#Index = 1) OR (#Index = 2) OR (#Index = 3));
   IF #_w1 THEN
       #previous_speed_tmpidx := #Index;
       #dint_tmp := #"InputTimeSpeed(time_each_pulse)";
       #real_tmp := DINT_TO_REAL(#dint_tmp);
       #real_tmp_1 := 60000.0/(#real_tmp*#number_of_gears_tmp);
       #real_tmp_2 := ROUND(#real_tmp_1);
       #speed_tmp[#Index] := REAL_TO_DINT(#real_tmp_2);
   END_IF;
END_REGION

REGION Network 4
   RUNG wire#powerrail
      Move(in := #dint_tmp, out1 => #"TimePerPulse(x1ms)")
   END_RUNG
   // the same network as SCL:
   #"TimePerPulse(x1ms)" := #dint_tmp;
END_REGION

REGION Network 5
   RUNG wire#powerrail
      { S7_Templates := "SrcType := Time" } GT_Contact(in1 := #"InputTimeSpeed(time_each_pulse)", in2 := T#0ms)
      wire#w1
      { S7_Templates := "SrcType := DInt" } EQ_Contact(in1 := #speed_tmp[1], in2 := #speed_tmp[2])
      wire#w2
      { S7_Templates := "SrcType := DInt" } EQ_Contact(in1 := #speed_tmp[1], in2 := #speed_tmp[3])
      wire#w3
      Move(in := #speed_tmp[1], out1 => #"OutputSpeed(rpm)")
   END_RUNG
   RUNG wire#w1
      Contact( "AlwaysTRUE" )
   END_RUNG wire#w2
   RUNG wire#w2
      Contact( "AlwaysTRUE" )
   END_RUNG wire#w3
   // the same network as SCL:
   IF (#"InputTimeSpeed(time_each_pulse)" > T#0ms) AND ((#speed_tmp[1] = #speed_tmp[2]) OR "AlwaysTRUE") AND ((#speed_tmp[1] = #speed_tmp[3]) OR "AlwaysTRUE") THEN
       #"OutputSpeed(rpm)" := #speed_tmp[1];
   END_IF;
END_REGION
END_FUNCTION_BLOCK

FUNCTION_BLOCK "1.3 Speed Interrupt"   // FB2, LAD
{ S7_Optimized_Access := 'TRUE' }
VERSION : 0.1
   VAR_OUTPUT
      TimeSpeed : Time;
      speed_tmpidx : Int;
   END_VAR
   VAR RETAIN
      ".IEC_TIMER_SensorSpeed" : IEC_TIMER;
      bSpeedStart : Bool;
   END_VAR
BEGIN

REGION Network 1
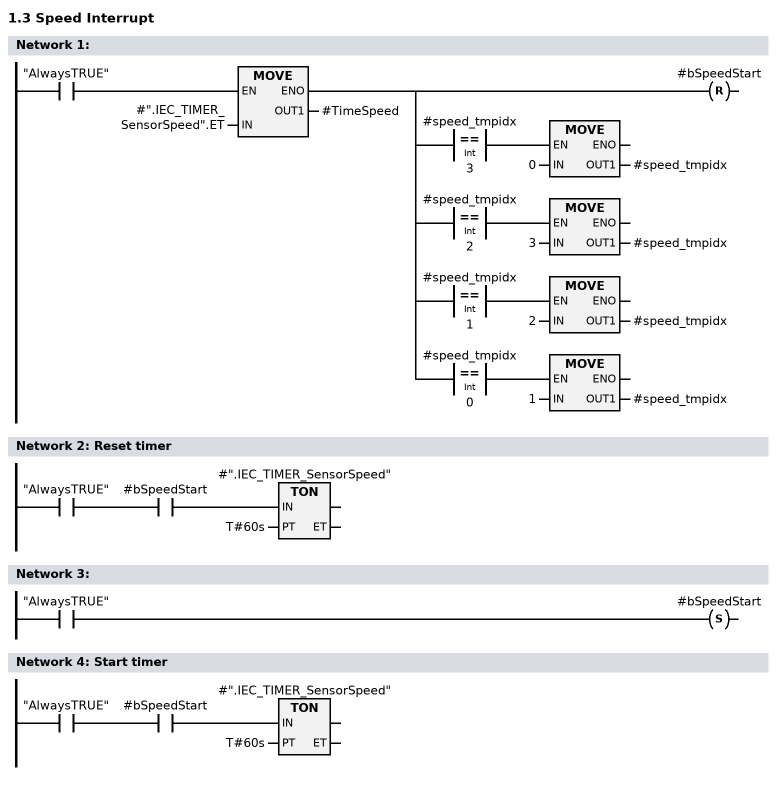
   RUNG wire#powerrail
      Contact( "AlwaysTRUE" )
      Move(in := #".IEC_TIMER_SensorSpeed".ET, out1 => #TimeSpeed)
      wire#w1
      R_Coil( #bSpeedStart )
   END_RUNG
   RUNG wire#w1
      { S7_Templates := "SrcType := Int" } EQ_Contact(in1 := #speed_tmpidx, in2 := 3)
      Move(in := 0, out1 => #speed_tmpidx)
   END_RUNG
   RUNG wire#w1
      { S7_Templates := "SrcType := Int" } EQ_Contact(in1 := #speed_tmpidx, in2 := 2)
      Move(in := 3, out1 => #speed_tmpidx)
   END_RUNG
   RUNG wire#w1
      { S7_Templates := "SrcType := Int" } EQ_Contact(in1 := #speed_tmpidx, in2 := 1)
      Move(in := 2, out1 => #speed_tmpidx)
   END_RUNG
   RUNG wire#w1
      { S7_Templates := "SrcType := Int" } EQ_Contact(in1 := #speed_tmpidx, in2 := 0)
      Move(in := 1, out1 => #speed_tmpidx)
   END_RUNG
   // the same network as SCL:
   IF "AlwaysTRUE" THEN
       #TimeSpeed := #".IEC_TIMER_SensorSpeed".ET;
       #bSpeedStart := FALSE;
   END_IF;
   IF "AlwaysTRUE" AND (#speed_tmpidx = 3) THEN #speed_tmpidx := 0; END_IF;
   IF "AlwaysTRUE" AND (#speed_tmpidx = 2) THEN #speed_tmpidx := 3; END_IF;
   IF "AlwaysTRUE" AND (#speed_tmpidx = 1) THEN #speed_tmpidx := 2; END_IF;
   IF "AlwaysTRUE" AND (#speed_tmpidx = 0) THEN #speed_tmpidx := 1; END_IF;
END_REGION

REGION Network 2: Reset timer
   #".IEC_TIMER_SensorSpeed".TON(IN := "AlwaysTRUE" AND #bSpeedStart, PT := T#60s);
END_REGION

REGION Network 3
   RUNG wire#powerrail
      Contact( "AlwaysTRUE" )
      S_Coil( #bSpeedStart )
   END_RUNG
   // the same network as SCL:
   IF "AlwaysTRUE" THEN #bSpeedStart := TRUE; END_IF;
END_REGION

REGION Network 4: Start timer
   #".IEC_TIMER_SensorSpeed".TON(IN := "AlwaysTRUE" AND #bSpeedStart, PT := T#60s);
END_REGION
END_FUNCTION_BLOCK

FUNCTION_BLOCK "Speed_Sensor"   // FB6, LAD
{ S7_Optimized_Access := 'TRUE' }
VERSION : 0.1
   VAR_INPUT
      "InputTimeSpeed(time_each_pulse)" : Time;
      NumberOfGears : UInt;
      Gear : DInt;
   END_VAR
   VAR_OUTPUT
      "TimePerPulse(x1ms)" : DInt;
      "OutputSpeedMeasure(rpm)" : DInt;
      "OutputSpeedMotor(rpm)" : DInt;
   END_VAR
   VAR_IN_OUT
      speed_array : Array[1..50] of Real;
      index_array : USInt;
   END_VAR
   VAR_TEMP
      number_of_gears_tmp : Real;
      dint_tmp : DInt;
      real_tmp : Real;
      speed_real : Real;
      gear_tmp : Real;
      speed_motor_tmp : Real;
      speed_motor_avg_tmp : Real;
      speed_motor_avg_tmp_dint : DInt;
   END_VAR
   VAR_TEMP   // added for the SCL form of the ladder/FBD networks
      _w1 : Bool;
   END_VAR
BEGIN

REGION Network 1
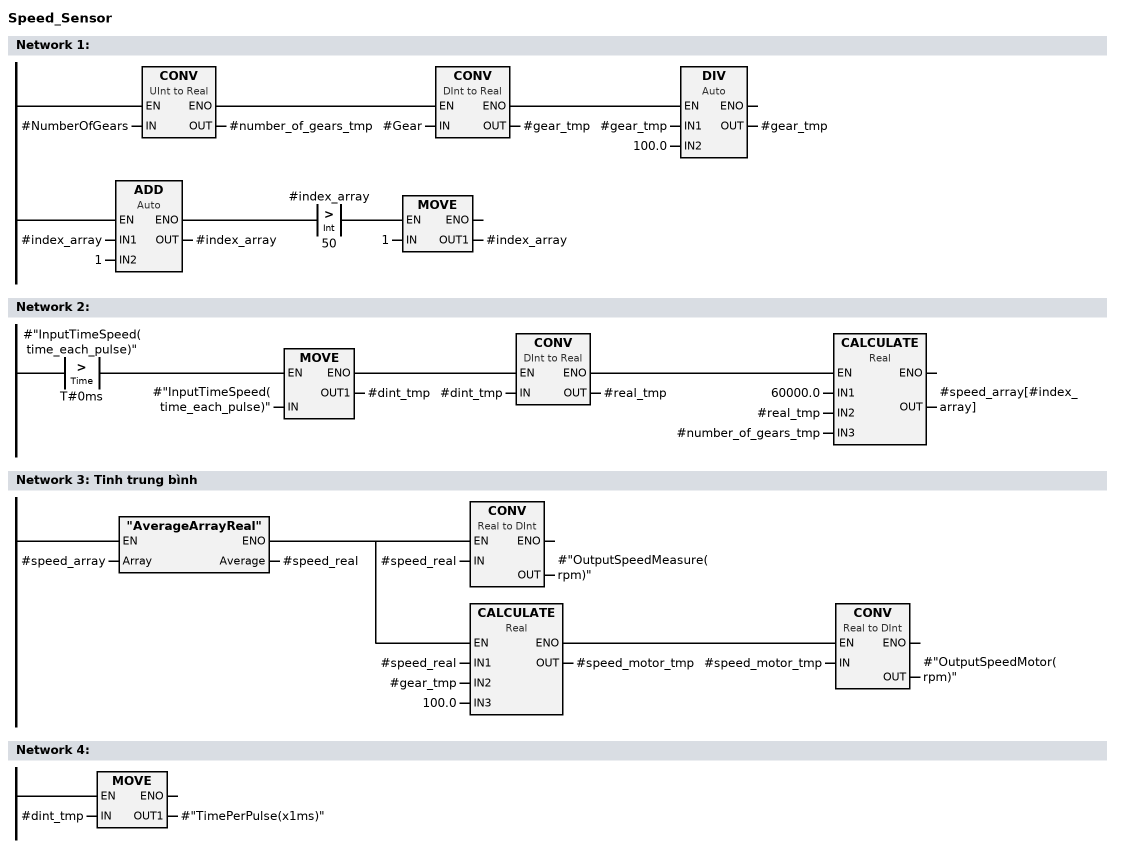
   RUNG wire#powerrail
      { S7_Templates := "[SrcType := UInt, DestType := Real]" } Convert(in := #NumberOfGears, out => #number_of_gears_tmp)
      { S7_Templates := "[SrcType := DInt, DestType := Real]" } Convert(in := #Gear, out => #gear_tmp)
      Div(in1 := #gear_tmp, in2 := 100.0, out => #gear_tmp)
   END_RUNG
   RUNG wire#powerrail
      Add(in1 := #index_array, in2 := 1, out => #index_array)
      { S7_Templates := "SrcType := Int" } GT_Contact(in1 := #index_array, in2 := 50)
      Move(in := 1, out1 => #index_array)
   END_RUNG
   // the same network as SCL:
   #number_of_gears_tmp := UINT_TO_REAL(#NumberOfGears);
   #gear_tmp := DINT_TO_REAL(#Gear);
   #gear_tmp := #gear_tmp / 100.0;
   #index_array := #index_array + 1;
   IF #index_array > 50 THEN #index_array := 1; END_IF;
END_REGION

REGION Network 2
   RUNG wire#powerrail
      { S7_Templates := "SrcType := Time" } GT_Contact(in1 := #"InputTimeSpeed(time_each_pulse)", in2 := T#0ms)
      Move(in := #"InputTimeSpeed(time_each_pulse)", out1 => #dint_tmp)
      { S7_Templates := "[SrcType := DInt, DestType := Real]" } Convert(in := #dint_tmp, out => #real_tmp)
      { S7_Templates := "SrcType := Real"; S7_Expression := "IN1/(IN2*IN3)" } Calculate(in1 := 60000.0, in2 := #real_tmp, in3 := #number_of_gears_tmp, out => #speed_array[#index_array])
   END_RUNG
   // the same network as SCL:
   IF #"InputTimeSpeed(time_each_pulse)" > T#0ms THEN
       #dint_tmp := #"InputTimeSpeed(time_each_pulse)";
       #real_tmp := DINT_TO_REAL(#dint_tmp);
       #speed_array[#index_array] := 60000.0/(#real_tmp*#number_of_gears_tmp);
   END_IF;
END_REGION

REGION Network 3: Tinh trung bình
   RUNG wire#powerrail
      "AverageArrayReal"("Array" := #speed_array, Average => #speed_real)
      wire#w1
      { S7_Templates := "[SrcType := Real, DestType := DInt]" } Convert(in := #speed_real, out => #"OutputSpeedMeasure(rpm)")
   END_RUNG
   RUNG wire#w1
      { S7_Templates := "SrcType := Real"; S7_Expression := "IN1*IN2*IN3" } Calculate(in1 := #speed_real, in2 := #gear_tmp, in3 := 100.0, out => #speed_motor_tmp)
      { S7_Templates := "[SrcType := Real, DestType := DInt]" } Convert(in := #speed_motor_tmp, out => #"OutputSpeedMotor(rpm)")
   END_RUNG
   // the same network as SCL:
   "AverageArrayReal"("Array" := #speed_array, Average => #speed_real, ENO => #_w1);
   IF #_w1 THEN
       #"OutputSpeedMeasure(rpm)" := REAL_TO_DINT(#speed_real);
       #speed_motor_tmp := #speed_real*#gear_tmp*100.0;
       #"OutputSpeedMotor(rpm)" := REAL_TO_DINT(#speed_motor_tmp);
   END_IF;
END_REGION

REGION Network 4
   RUNG wire#powerrail
      Move(in := #dint_tmp, out1 => #"TimePerPulse(x1ms)")
   END_RUNG
   // the same network as SCL:
   #"TimePerPulse(x1ms)" := #dint_tmp;
END_REGION
END_FUNCTION_BLOCK

FUNCTION "CalculatorSpeed" : Void   // FC60, SCL
{ S7_Optimized_Access := 'TRUE' }
VERSION : 0.1
   VAR_INPUT
      PPR : UInt;
      "SampleTime(x1ms)" : UInt;
      Coef : UInt;
   END_VAR
   VAR_OUTPUT
      RPM : DInt;
   END_VAR
   VAR_IN_OUT
      Pulses : UInt;
   END_VAR
   VAR_TEMP
      rounds_ms : Real;
      "number _of_rounds" : Real;
   END_VAR
   VAR CONSTANT
      ms_to_minute : UInt := 60000;
   END_VAR
BEGIN
   IF #"SampleTime(x1ms)">0 THEN
       #"number _of_rounds" := UINT_TO_REAL(#Pulses) / UINT_TO_REAL(#PPR);
       #rounds_ms := #"number _of_rounds" / UINT_TO_REAL(#"SampleTime(x1ms)");
       #Pulses := 0;
   ELSE
       #rounds_ms := 0;
   END_IF;

   #RPM := REAL_TO_DINT(#rounds_ms * #ms_to_minute * #Coef);
END_FUNCTION

FUNCTION "AverageArrayReal" : Void   // FC67, SCL
{ S7_Optimized_Access := 'TRUE' }
VERSION : 0.1
   VAR_INPUT
      "Array" : Array[1..50] of Real;
   END_VAR
   VAR_OUTPUT
      Average : Real;
   END_VAR
   VAR_TEMP
      index : USInt;
      value_tmp : Real;
   END_VAR
BEGIN
   FOR #index := 1 TO 50 DO
       #value_tmp += #Array[#index];
   END_FOR;

   #Average := #value_tmp / 50.0;
END_FUNCTION

// folder: Sensor-StartStop

FUNCTION_BLOCK "StartStop"   // FB5, LAD
{ S7_Optimized_Access := 'TRUE' }
VERSION : 0.1
   VAR_INPUT
      bStartStopTrigger : Bool;
      TonFilter_x1ms : UInt := 10;   // x1ms
      ToffFilter_x1ms : UInt := 10;   // x1ms
   END_VAR
   VAR_OUTPUT
      bOutput : Bool;
   END_VAR
   VAR
      TimerTon : Time;
      TimerToff : Time;
   END_VAR
   VAR RETAIN
      P_tmp : Bool;
   END_VAR
   VAR
      Ton_start : Bool;
   END_VAR
   VAR RETAIN
      IEC_Ton : IEC_TIMER;
      IEC_Toff : IEC_TIMER;
      N_tmp : Bool;
   END_VAR
   VAR
      Toff_start : Bool;
   END_VAR
   VAR_TEMP   // added for the SCL form of the ladder/FBD networks
      _w1 : Bool;
   END_VAR
BEGIN

REGION Network 1
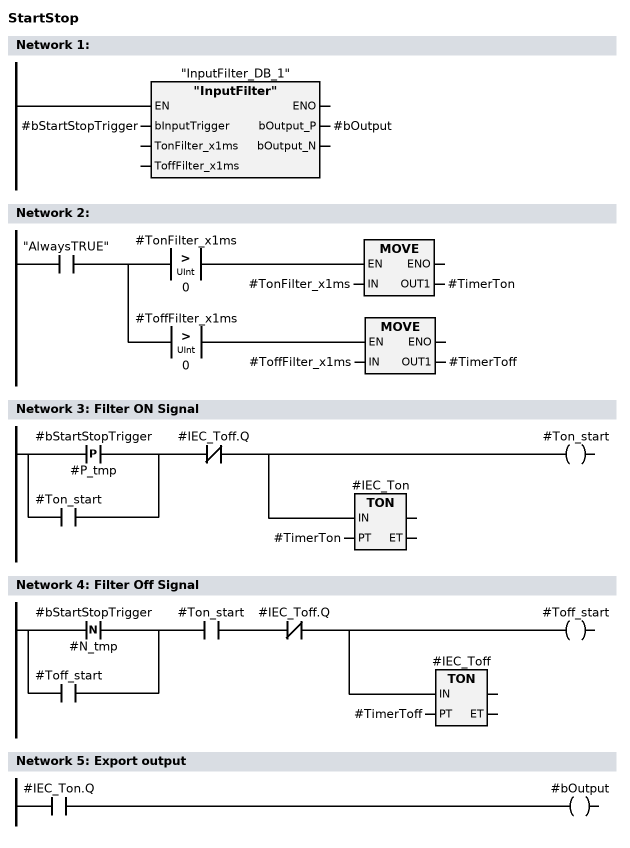
   RUNG wire#powerrail
      "InputFilter_DB_1"(bInputTrigger := #bStartStopTrigger, TonFilter_x1ms :=, ToffFilter_x1ms :=, bOutput_P => #bOutput, bOutput_N =>)
   END_RUNG
   // the same network as SCL:
   "InputFilter_DB_1"(bInputTrigger := #bStartStopTrigger, bOutput_P => #bOutput);   // "InputFilter"
END_REGION

REGION Network 2
   RUNG wire#powerrail
      Contact( "AlwaysTRUE" )
      wire#w1
      { S7_Templates := "SrcType := UInt" } GT_Contact(in1 := #TonFilter_x1ms, in2 := 0)
      Move(in := #TonFilter_x1ms, out1 => #TimerTon)
   END_RUNG
   RUNG wire#w1
      { S7_Templates := "SrcType := UInt" } GT_Contact(in1 := #ToffFilter_x1ms, in2 := 0)
      Move(in := #ToffFilter_x1ms, out1 => #TimerToff)
   END_RUNG
   // the same network as SCL:
   IF "AlwaysTRUE" AND (#TonFilter_x1ms > 0) THEN #TimerTon := #TonFilter_x1ms; END_IF;
   IF "AlwaysTRUE" AND (#ToffFilter_x1ms > 0) THEN #TimerToff := #ToffFilter_x1ms; END_IF;
END_REGION

REGION Network 3: Filter ON Signal
   #_w1 := #bStartStopTrigger AND NOT #P_tmp;   // rising edge of #bStartStopTrigger
   #P_tmp := #bStartStopTrigger;
   #Ton_start := (#_w1 OR #Ton_start) AND NOT #IEC_Toff.Q;
   #IEC_Ton.TON(IN := #Ton_start, PT := #TimerTon);
END_REGION

REGION Network 4: Filter Off Signal
   #_w1 := NOT #bStartStopTrigger AND #N_tmp;   // falling edge of #bStartStopTrigger
   #N_tmp := #bStartStopTrigger;
   #Toff_start := (#_w1 OR #Toff_start) AND #Ton_start AND NOT #IEC_Toff.Q;
   #IEC_Toff.TON(IN := #Toff_start, PT := #TimerToff);
END_REGION

REGION Network 5: Export output
   RUNG wire#powerrail
      Contact( #IEC_Ton.Q )
      Coil( #bOutput )
   END_RUNG
   // the same network as SCL:
   #bOutput := #IEC_Ton.Q;
END_REGION
END_FUNCTION_BLOCK

// folder: Server

FUNCTION_BLOCK "CheckConnectPLCServer"   // FB8, LAD
{ S7_Optimized_Access := 'TRUE' }
VERSION : 0.1
   VAR_INPUT
      Signal : Bool;
      "Timeout(s)" : USInt;
   END_VAR
   VAR_OUTPUT
      Status : Bool;
   END_VAR
   VAR
      IEC_Timer_0_Instance : TON_TIME;
      TagSignalN : Bool;
   END_VAR
   VAR_TEMP
      TimeOut : Time;
   END_VAR
   VAR_TEMP   // added for the SCL form of the ladder/FBD networks
      _w1 : Bool;
   END_VAR
BEGIN

REGION Network 1
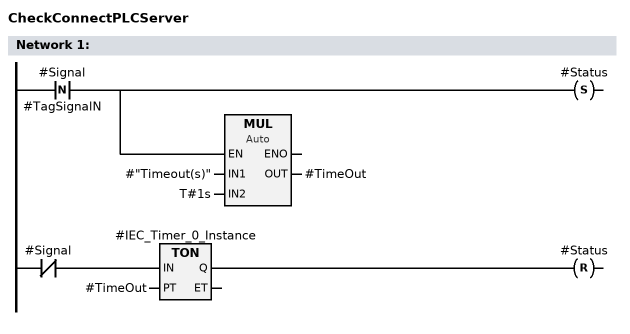
   #_w1 := NOT #Signal AND #TagSignalN;   // falling edge of #Signal
   #TagSignalN := #Signal;
   IF #_w1 THEN
       #Status := TRUE;
       #TimeOut := #"Timeout(s)" * T#1s;
   END_IF;
   #IEC_Timer_0_Instance(IN := NOT #Signal, PT := #TimeOut);   // TON
   IF #IEC_Timer_0_Instance.Q THEN #Status := FALSE; END_IF;
END_REGION
END_FUNCTION_BLOCK

// folder: Setting

FUNCTION "SettingInformation" : Void   // FC43, SCL
{ S7_Optimized_Access := 'TRUE' }
VERSION : 0.1
   VAR_IN_OUT
      event_confirm : Bool;
      event_cancel : Bool;
   END_VAR
BEGIN
   IF #event_confirm=TRUE THEN
       "DataSetting".InforStation.MachineCode := "DB_DataHMI".InforStation.MachineCode;

       #event_confirm := FALSE;

       "DB_Server".SyncSettings := 1;
   END_IF;

   IF #event_cancel = TRUE THEN
       "DB_DataHMI".InforStation.MachineCode:="DataSetting".InforStation.MachineCode;

       #event_cancel := FALSE;
   END_IF;
END_FUNCTION

FUNCTION "SettingGeneral" : Void   // FC44, SCL
{ S7_Optimized_Access := 'TRUE' }
VERSION : 0.1
   VAR_IN_OUT
      event_confirm : Bool;
      event_cancel : Bool;
   END_VAR
BEGIN
   IF #event_confirm = TRUE THEN
       "DataSetting"."CounterFilterOn(ms)" := "DB_DataHMI"."CounterFilterOn(ms)";
       "DataSetting"."CounterFilterOff(ms)" := "DB_DataHMI"."CounterFilterOff(ms)";
       "DataSetting"."TimeThresholdLoss(ms)" := "DB_DataHMI"."TimeThresholdLoss(ms)";
       "DataSetting"."TimeThresholdShowWarningAssignLoss(s)" := "DB_DataHMI"."TimeThresholdShowWarningAssignLoss(s)";

       #event_confirm := FALSE;

       "DB_Server".SyncSettings := 1;
   END_IF;

   IF #event_cancel = TRUE THEN
       "DB_DataHMI"."CounterFilterOn(ms)":="DataSetting"."CounterFilterOn(ms)";
       "DB_DataHMI"."CounterFilterOff(ms)":="DataSetting"."CounterFilterOff(ms)";
       "DB_DataHMI"."TimeThresholdLoss(ms)":="DataSetting"."TimeThresholdLoss(ms)";
       "DB_DataHMI"."TimeThresholdShowWarningAssignLoss(s)":="DataSetting"."TimeThresholdShowWarningAssignLoss(s)";

       #event_cancel := FALSE;
   END_IF;
END_FUNCTION

FUNCTION "SettingBladeTemperature" : Void   // FC45, SCL
{ S7_Optimized_Access := 'TRUE' }
VERSION : 0.1
   VAR_IN_OUT
      event_confirm : Bool;
      event_cancel : Bool;
   END_VAR
BEGIN
   // IF #event_confirm = TRUE THEN
   //     "DataSetting".SettingBladeTemp := "DB_DataHMI".SensorBladeTemp;

   //     #event_confirm := FALSE;

   //     "DB_Server".SyncSettings := 1;
   // END_IF;

   // IF #event_cancel = TRUE THEN
   //     "DB_DataHMI".SensorBladeTemp := "DataSetting".SettingBladeTemp;

   //     #event_cancel := FALSE;
   // END_IF;
END_FUNCTION

FUNCTION "SettingCurrent" : Void   // FC46, SCL
{ S7_Optimized_Access := 'TRUE' }
VERSION : 0.1
   VAR_IN_OUT
      event_confirm : Bool;
      event_cancel : Bool;
   END_VAR
BEGIN
   // IF #event_confirm = TRUE THEN
   //     "DataSetting".SettingCurrent := "DB_DataHMI".SensorCurrent;

   //     #event_confirm := FALSE;

   //     "DB_Server".SyncSettings := 1;
   // END_IF;

   // IF #event_cancel = TRUE THEN
   //     "DB_DataHMI".SensorCurrent := "DataSetting".SettingCurrent;

   //     #event_cancel := FALSE;
   // END_IF;
END_FUNCTION

FUNCTION "SettingSpeed" : Void   // FC47, SCL
{ S7_Optimized_Access := 'TRUE' }
VERSION : 0.1
   VAR_IN_OUT
      event_confirm : Bool;
      event_cancel : Bool;
   END_VAR
BEGIN
   // IF #event_confirm = TRUE THEN
   //     "DataSetting".SettingWheelSpeed := "DB_DataHMI".SensorWheelSpeed;

   //     #event_confirm := FALSE;

   //     "DB_Server".SyncSettings := 1;
   // END_IF;

   // IF #event_cancel = TRUE THEN
   //     "DB_DataHMI".SensorWheelSpeed := "DataSetting".SettingWheelSpeed;

   //     #event_cancel := FALSE;
   // END_IF;
END_FUNCTION

FUNCTION "SettingPressureForce" : Void   // FC48, SCL
{ S7_Optimized_Access := 'TRUE' }
VERSION : 0.1
   VAR_IN_OUT
      event_confirm : Bool;
      event_cancel : Bool;
   END_VAR
BEGIN
   IF #event_confirm = TRUE THEN
       // "DataSetting".SettingForce := "DB_DataHMI".Force;
       // "DataSetting".SensorPresureIn := "DB_DataHMI".SensorPresureIn;
       // "DataSetting".SensorPresureOut := "DB_DataHMI".SensorPresureOut;
       #event_confirm := FALSE;

       "DB_Server".SyncSettings := 1;
   END_IF;

   IF #event_cancel = TRUE THEN
       // "DB_DataHMI".Force := "DataSetting".SettingForce;
       // "DB_DataHMI".SensorPresureIn := "DataSetting".SensorPresureIn;
       // "DB_DataHMI".SensorPresureOut := "DataSetting".SensorPresureOut;
       #event_cancel := FALSE;
   END_IF;
END_FUNCTION

FUNCTION "MoveDataSettingToHmi" : Void   // FC49, SCL
{ S7_Optimized_Access := 'TRUE' }
VERSION : 0.1
BEGIN
   //Information
   "DB_DataHMI".InforStation := "DataSetting".InforStation;

   //General
   "DB_DataHMI"."CounterFilterOn(ms)" := "DataSetting"."CounterFilterOn(ms)";
   "DB_DataHMI"."CounterFilterOff(ms)" := "DataSetting"."CounterFilterOff(ms)";
   "DB_DataHMI"."TimeThresholdLoss(ms)" := "DataSetting"."TimeThresholdLoss(ms)";
   "DB_DataHMI"."TimeThresholdClearBlade(ms)" := "DataSetting"."TimeThresholdClearBlade(ms)";
   "DB_DataHMI"."TimeThresholdShowWarningAssignLoss(s)" := "DataSetting"."TimeThresholdShowWarningAssignLoss(s)";

   //Blade Temperature
   "DB_DataHMI".BladeTemperature.Common := "DataSetting".SettingBladeTemp;

   //Current
   "DB_DataHMI".Current.Common := "DataSetting".SettingCurrent;

   //Speed
   "DB_DataHMI".WheelSpeed.Common := "DataSetting".SettingWheelSpeed;

   //PresureIn
   "DB_DataHMI".PressureIn.Common := "DataSetting".SettingPresureIn;

   //PresureOut
   "DB_DataHMI".PressureOut.Common := "DataSetting".SettingPresureOut;

   //Force
   "DB_DataHMI".ForceXilanh.Common := "DataSetting".SettingForceXilanh;

   //Độ phân giải
   "DB_DataHMI".AnalogSensorMin := "DB_Machine".AnalogSensorMin;
   "DB_DataHMI".AnalogSensorMax := "DB_Machine".AnalogSensorMax;
END_FUNCTION

FUNCTION "MoveDataSettingToServer" : Void   // FC50, SCL
{ S7_Optimized_Access := 'TRUE' }
VERSION : 0.1
BEGIN
   //Setting Infor
   "DB_Server".InforStation := "DataSetting".InforStation;

   //General
   "DB_Server"."CounterFilterOn(ms)" := "DataSetting"."CounterFilterOn(ms)";
   "DB_Server"."CounterFilterOff(ms)" := "DataSetting"."CounterFilterOff(ms)";
   "DB_Server"."TimeThresholdLoss(ms)" := "DataSetting"."TimeThresholdLoss(ms)";
   "DB_Server"."TimeThresholdShowWarningAssignLoss(s)" := "DataSetting"."TimeThresholdShowWarningAssignLoss(s)";

   //Blade Temperature
   "DB_Server".SettingBladeTemp."RangeMinSensor(x100)":="DataSetting".SettingBladeTemp."RangMinSensor(x100)";
   "DB_Server".SettingBladeTemp."RangeMaxSensor(x100)" := "DataSetting".SettingBladeTemp."RangMaxSensor(x100)";
   "DB_Server".SettingBladeTemp."Offset(x100)" := "DataSetting".SettingBladeTemp."Offset(x100)";

   "DB_Server".SettingBladeTemp."Upper(x100)" := "DataSetting".SettingBladeTemp."SettingUpper(x100)";
   "DB_Server".SettingBladeTemp."Lower(x100)" := "DataSetting".SettingBladeTemp."SettingLower(x100)";


   //Current
   "DB_Server".SettingCurrent."RangeMinSensor(x100)" := "DataSetting".SettingCurrent."RangMinSensor(x100)";
   "DB_Server".SettingCurrent."RangeMaxSensor(x100)" := "DataSetting".SettingCurrent."RangMaxSensor(x100)";
   "DB_Server".SettingCurrent."Offset(x100)" := "DataSetting".SettingCurrent."Offset(x100)";

   "DB_Server".SettingCurrent."Upper(x100)" := "DataSetting".SettingCurrent."SettingUpper(x100)";
   "DB_Server".SettingCurrent."Lower(x100)" := "DataSetting".SettingCurrent."SettingLower(x100)";

   //Speed
   "DB_Server".SettingWheelSpeed.Infor."Lower(x100)" := "DataSetting".SettingWheelSpeed."SettingLower(x100)";
   "DB_Server".SettingWheelSpeed.Infor."Upper(x100)" := "DataSetting".SettingWheelSpeed."SettingUpper(x100)";
   "DB_Server".SettingWheelSpeed.Infor."Offset(x100)" := "DataSetting".SettingWheelSpeed."Offset(x100)";

   "DB_Server".SettingWheelSpeed."GearRatio(x100)" := "DataSetting".SettingWheelSpeed."GearRatio(x100)";
   "DB_Server".SettingWheelSpeed.NumberOfGears := "DataSetting".SettingWheelSpeed.NumberOfGears;


   //Pressure
   "DB_Server".SensorPresureOut."RangeMinSensor(x100)" := "DataSetting".SettingWheelSpeed."SettingLower(x100)";
   "DB_Server".SensorPresureOut."RangeMaxSensor(x100)" := "DataSetting".SettingWheelSpeed."SettingUpper(x100)";

   "DB_Server".SensorPresureOut."Lower(x100)" := "DataSetting".SettingPresureOut."SettingLower(x100)";
   "DB_Server".SensorPresureOut."Upper(x100)" := "DataSetting".SettingPresureOut."SettingUpper(x100)";

   //Force Xi lanh
   "DB_Server".SettingForce.Infor."Lower(x100)" := "DataSetting".SettingForceXilanh."SettingLower(x100)";
   "DB_Server".SettingForce.Infor."Upper(x100)" := "DataSetting".SettingForceXilanh."SettingUpper(x100)";
   "DB_Server".SettingForce.Infor."Offset(x100)" := "DataSetting".SettingForceXilanh."Offset(x100)";

   "DB_Server".SettingForce.Area := "DataSetting".SettingForceXilanh."Area(cm2 x 100)";
   "DB_Server".SettingForce."CoefficientUnit(x100)" := "DataSetting".SettingForceXilanh."CoefficientUnit(x100)";
END_FUNCTION

FUNCTION "SyncSettingServer" : Void   // FC58, SCL
{ S7_Optimized_Access := 'TRUE' }
VERSION : 0.1
BEGIN
   //Đợi Web code để biết gửi những gì
   //Temperature
   "DataSetting".SettingBladeTemp."SettingLower(x100)" := "DB_Server".SettingBladeTemp."Lower(x100)";
   "DataSetting".SettingBladeTemp."SettingUpper(x100)" := "DB_Server".SettingBladeTemp."Upper(x100)";

   //Current
   "DataSetting".SettingCurrent."SettingLower(x100)" := "DB_Server".SettingCurrent."Lower(x100)";
   "DataSetting".SettingCurrent."SettingUpper(x100)" := "DB_Server".SettingCurrent."Upper(x100)";

   //Speed
   "DataSetting".SettingWheelSpeed."SettingLower(x100)" := "DB_Server".SettingWheelSpeed.Infor."Lower(x100)";
   "DataSetting".SettingWheelSpeed."SettingUpper(x100)" := "DB_Server".SettingWheelSpeed.Infor."Upper(x100)";

   //Pressure Out
   "DataSetting".SettingPresureOut."SettingLower(x100)" := "DB_Server".SensorPresureOut."Lower(x100)";
   "DataSetting".SettingPresureOut."SettingUpper(x100)" :=  "DB_Server".SensorPresureOut."Upper(x100)";

   //Giá trị cài đặt qua HMI
   "DB_DataHMI".BladeTemperature.Common := "DataSetting".SettingBladeTemp;
   "DB_DataHMI".Current.Common := "DataSetting".SettingCurrent;
   "DB_DataHMI".PressureOut.Common := "DataSetting".SettingPresureOut;
   "DB_DataHMI".WheelSpeed.Common := "DataSetting".SettingWheelSpeed;


   "DB_Server".SyncSettings := 3;
END_FUNCTION

FUNCTION "SaveSettingHMI" : Void   // FC61, SCL
{ S7_Optimized_Access := 'TRUE' }
VERSION : 0.1
   VAR_IN_OUT
      Confirm : Bool;
      Cancel : Bool;
      IndexTabSetting : Int;
      "Return value = 1" : USInt;
   END_VAR
BEGIN
   IF #Confirm=TRUE OR #Cancel=TRUE THEN
       IF #Confirm = TRUE THEN
           CASE #IndexTabSetting OF
               1: //Information 
                   "DataSetting".InforStation := "DB_DataHMI".InforStation;

                   //Server
                   "DB_Server".InforStation := "DB_DataHMI".InforStation;

                   //Bit Show Thông báo
                   "DB_DataHMI".EventBitShowSaveSettingSuccess := TRUE;
               2: // General
                   "DataSetting"."CounterFilterOff(ms)" := "DB_DataHMI"."CounterFilterOff(ms)";
                   "DataSetting"."CounterFilterOn(ms)" := "DB_DataHMI"."CounterFilterOn(ms)";
                   "DataSetting"."TimeThresholdLoss(ms)" := "DB_DataHMI"."TimeThresholdLoss(ms)";
                   "DataSetting"."TimeThresholdClearBlade(ms)" := "DB_DataHMI"."TimeThresholdClearBlade(ms)";
                   "DataSetting"."TimeThresholdShowWarningAssignLoss(s)" := "DB_DataHMI"."TimeThresholdShowWarningAssignLoss(s)";

                   //Server
                   "DB_Server"."CounterFilterOff(ms)" := "DB_DataHMI"."CounterFilterOff(ms)";
                   "DB_Server"."CounterFilterOn(ms)" := "DB_DataHMI"."CounterFilterOn(ms)";
                   "DB_Server"."TimeThresholdLoss(ms)" := "DB_DataHMI"."TimeThresholdLoss(ms)";
                   "DB_Server"."TimeThresholdBlade(ms)" := "DB_DataHMI"."TimeThresholdClearBlade(ms)";
                   "DB_Server"."TimeThresholdShowWarningAssignLoss(s)" := "DB_DataHMI"."TimeThresholdShowWarningAssignLoss(s)";

                   //Bit Show Thông báo
                   "DB_DataHMI".EventBitShowSaveSettingSuccess := TRUE;
               3: // Blade Temperature
                   "DataSetting".SettingBladeTemp := "DB_DataHMI".BladeTemperature.Common;
                   "Analogs_DB".Temperature.MinRealScale := "DB_DataHMI".BladeTemperature.Common."RangMinSensor(x100)";
                   "Analogs_DB".Temperature.MaxRealScale := "DB_DataHMI".BladeTemperature.Common."RangMaxSensor(x100)";

                   //Server
                   "DB_Server".SettingBladeTemp."RangeMinSensor(x100)" := "DataSetting".SettingBladeTemp."RangMinSensor(x100)";
                   "DB_Server".SettingBladeTemp."RangeMaxSensor(x100)" := "DataSetting".SettingBladeTemp."RangMaxSensor(x100)";
                   "DB_Server".SettingBladeTemp."Offset(x100)" := "DataSetting".SettingBladeTemp."Offset(x100)";

                   "DB_Server".SettingBladeTemp."Upper(x100)" := "DataSetting".SettingBladeTemp."SettingUpper(x100)";
                   "DB_Server".SettingBladeTemp."Lower(x100)" := "DataSetting".SettingBladeTemp."SettingLower(x100)";

                   //Bit Show Thông báo
                   "DB_DataHMI".EventBitShowSaveSettingSuccess := TRUE;
               4: //Curent
                   "DataSetting".SettingCurrent := "DB_DataHMI".Current.Common;
                   "Analogs_DB".Current.MinRealScale := "DB_DataHMI".Current.Common."RangMinSensor(x100)";
                   "Analogs_DB".Current.MaxRealScale := "DB_DataHMI".Current.Common."RangMaxSensor(x100)";

                   //Server
                   "DB_Server".SettingCurrent."RangeMinSensor(x100)" := "DataSetting".SettingCurrent."RangMinSensor(x100)";
                   "DB_Server".SettingCurrent."RangeMaxSensor(x100)" := "DataSetting".SettingCurrent."RangMaxSensor(x100)";
                   "DB_Server".SettingCurrent."Offset(x100)" := "DataSetting".SettingCurrent."Offset(x100)";

                   "DB_Server".SettingCurrent."Upper(x100)" := "DataSetting".SettingCurrent."SettingUpper(x100)";
                   "DB_Server".SettingCurrent."Lower(x100)" := "DataSetting".SettingCurrent."SettingLower(x100)";

                   //Bit Show Thông báo
                   "DB_DataHMI".EventBitShowSaveSettingSuccess := TRUE;
               5: //Speed
                   "DataSetting".SettingWheelSpeed := "DB_DataHMI".WheelSpeed.Common;

                   //Server
                   "DB_Server".SettingWheelSpeed.Infor."Lower(x100)" := "DataSetting".SettingWheelSpeed."SettingLower(x100)";
                   "DB_Server".SettingWheelSpeed.Infor."Upper(x100)" := "DataSetting".SettingWheelSpeed."SettingUpper(x100)";
                   "DB_Server".SettingWheelSpeed.Infor."Offset(x100)" := "DataSetting".SettingWheelSpeed."Offset(x100)";

                   "DB_Server".SettingWheelSpeed."GearRatio(x100)" := "DataSetting".SettingWheelSpeed."GearRatio(x100)";
                   "DB_Server".SettingWheelSpeed.NumberOfGears := "DataSetting".SettingWheelSpeed.NumberOfGears;

                   //Bit Show Thông báo
                   "DB_DataHMI".EventBitShowSaveSettingSuccess := TRUE;
               6: //Pressure
                   "DataSetting".SettingPresureOut := "DB_DataHMI".PressureOut.Common;


                   "Analogs_DB".Pressure_OUT.MinRealScale := "DB_DataHMI".PressureOut.Common."RangMinSensor(x100)";
                   "Analogs_DB".Pressure_OUT.MaxRealScale := "DB_DataHMI".PressureOut.Common."RangMaxSensor(x100)";



                   //Server
                   //Pressure
                   "DB_Server".SensorPresureOut."RangeMinSensor(x100)" := "DataSetting".SettingWheelSpeed."SettingLower(x100)";
                   "DB_Server".SensorPresureOut."RangeMaxSensor(x100)" := "DataSetting".SettingWheelSpeed."SettingUpper(x100)";

                   "DB_Server".SensorPresureOut."Upper(x100)" := "DataSetting".SettingPresureOut."SettingUpper(x100)";
                   "DB_Server".SensorPresureOut."Lower(x100)" := "DataSetting".SettingPresureOut."SettingLower(x100)";

                   //DB_Server".SettingForce."CoefficientUnit(x100)":="DataSetting".SettingForceXilanh."CoefficientUnit(x100)";
                   // //Force Xi lanh
                   // "DB_Server".SettingForce.Infor."Lower(x100)" := "DataSetting".SettingForceXilanh."SettingLower(x100)";
                   // "DB_Server".SettingForce.Infor."Upper(x100)" := "DataSetting".SettingForceXilanh."SettingUpper(x100)";
                   // "DB_Server".SettingForce.Infor."Offset(x100)" := "DataSetting".SettingForceXilanh."Offset(x100)";

                   // "DB_Server".SettingForce.Area := "DataSetting".SettingForceXilanh."Area(cm2 x 100)";
                   // "DB_Server".SettingForce."CoefficientUnit(x100)" := "DataSetting".SettingForceXilanh."CoefficientUnit(x100)";

                   //Bit Show Thông báo
                   "DB_DataHMI".EventBitShowSaveSettingSuccess := TRUE;
           END_CASE;
           #Confirm := FALSE;
           #"Return value = 1" := 1;
       END_IF;

       IF #Cancel = TRUE THEN
           CASE #IndexTabSetting OF
               1:
                   "DB_DataHMI".InforStation := "DataSetting".InforStation;
               2:
                   "DB_DataHMI"."CounterFilterOff(ms)" := "DataSetting"."CounterFilterOff(ms)";
                   "DB_DataHMI"."CounterFilterOn(ms)" := "DataSetting"."CounterFilterOn(ms)";
                   "DB_DataHMI"."TimeThresholdLoss(ms)" := "DataSetting"."TimeThresholdLoss(ms)";
                   "DB_DataHMI"."TimeThresholdShowWarningAssignLoss(s)" := "DataSetting"."TimeThresholdShowWarningAssignLoss(s)";
               3:
                   "DB_DataHMI".BladeTemperature.Common := "DataSetting".SettingBladeTemp;
               4:
                   "DB_DataHMI".Current.Common := "DataSetting".SettingCurrent;
               5:
                   "DB_DataHMI".WheelSpeed.Common := "DataSetting".SettingWheelSpeed;
               6:
                   "DB_DataHMI".PressureOut.Common := "DataSetting".SettingPresureOut;
                   "DB_DataHMI".ForceXilanh.Common := "DataSetting".SettingForceXilanh;
           END_CASE;
           #Cancel := FALSE;
       END_IF;
       #IndexTabSetting := 0;
   END_IF;
END_FUNCTION

FUNCTION "MoveDataSettingToBufferAnalog" : Void   // FC62, SCL
{ S7_Optimized_Access := 'TRUE' }
VERSION : 0.1
BEGIN
   (* Temperature *)
   "Analogs_DB".Temperature.MinRealScale := "DataSetting".SettingBladeTemp."RangMinSensor(x100)" / 100;// Min giá trị thực
   "Analogs_DB".Temperature.MaxRealScale := "DataSetting".SettingBladeTemp."RangMaxSensor(x100)" / 100;// Max giá trị thực
   "Analogs_DB".Temperature.digit := 2;//Hiển thị sau dấu chấm 2 đơn vị

   (* Electric current *)
   "Analogs_DB".Current.MinRealScale := "DataSetting".SettingCurrent."RangMinSensor(x100)" / 100;// Min giá trị thực
   "Analogs_DB".Current.MaxRealScale := "DataSetting".SettingCurrent."RangMaxSensor(x100)" / 100;// Max giá trị thực
   "Analogs_DB".Current.digit := 2; //Hiển thị sau dấu chấm 2 đơn vị

   (* Pressure IN *)
   "Analogs_DB".Pressure_IN.MinRealScale := "DataSetting".SettingPresureIn."RangMinSensor(x100)" / 100;// Min giá trị thực
   "Analogs_DB".Pressure_IN.MaxRealScale := "DataSetting".SettingPresureIn."RangMaxSensor(x100)" / 100;// Max giá trị thực
   "Analogs_DB".Pressure_IN.digit := 2; //Hiển thị sau dấu chấm 2 đơn vị

   (* Pressure OUT *)
   "Analogs_DB".Pressure_OUT.MinRealScale := DINT_TO_REAL("DataSetting".SettingPresureOut."RangMinSensor(x100)") / 100; // Min giá trị thực
   "Analogs_DB".Pressure_OUT.MaxRealScale := DINT_TO_REAL("DataSetting".SettingPresureOut."RangMaxSensor(x100)") / 100; // Max giá trị thực
   "Analogs_DB".Pressure_OUT.digit := 2; //Hiển thị sau dấu chấm 2 đơn vị
END_FUNCTION

// folder: Simulation

FUNCTION_BLOCK "CreatePulse"   // FB9, LAD
{ S7_Optimized_Access := 'TRUE' }
VERSION : 0.1
   VAR_INPUT
      "pulse_on(x1ms)" : UInt;
      "pulse_off(x1ms)" : UInt;
   END_VAR
   VAR_OUTPUT
      pulse : Bool;
   END_VAR
   VAR
      IEC_Timer_0_Instance : TON_TIME;
      IEC_Timer_0_Instance_1 : TON_TIME;
   END_VAR
   VAR_TEMP
      time_on : Time;
      time_off : Time;
   END_VAR
BEGIN

REGION Network 1
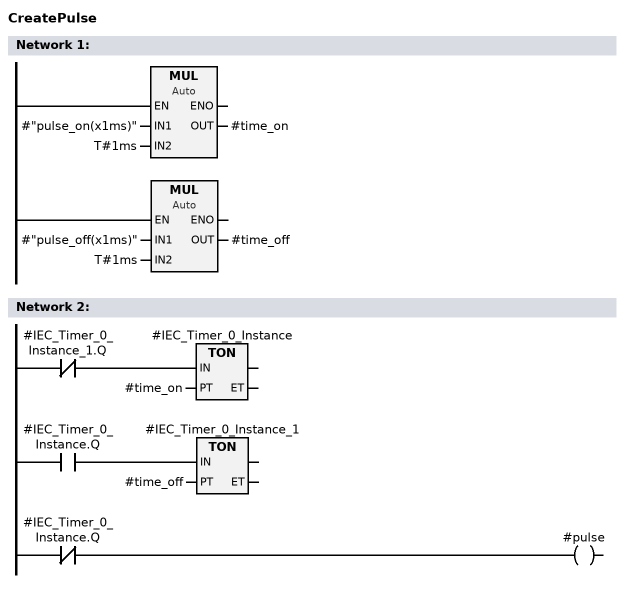
   RUNG wire#powerrail
      Mul(in1 := #"pulse_on(x1ms)", in2 := T#1ms, out => #time_on)
   END_RUNG
   RUNG wire#powerrail
      Mul(in1 := #"pulse_off(x1ms)", in2 := T#1ms, out => #time_off)
   END_RUNG
   // the same network as SCL:
   #time_on := #"pulse_on(x1ms)" * T#1ms;
   #time_off := #"pulse_off(x1ms)" * T#1ms;
END_REGION

REGION Network 2
   #IEC_Timer_0_Instance(IN := NOT #IEC_Timer_0_Instance_1.Q, PT := #time_on);   // TON
   #IEC_Timer_0_Instance_1(IN := #IEC_Timer_0_Instance.Q, PT := #time_off);   // TON
   #pulse := NOT #IEC_Timer_0_Instance.Q;
END_REGION
END_FUNCTION_BLOCK

FUNCTION "0.3 ClockSensorOutput" : Void   // FC2, LAD
{ S7_Optimized_Access := 'TRUE' }
VERSION : 0.1
   VAR_INPUT
      Index : Int;
      Clock_x10ms : UInt;
   END_VAR
   VAR_OUTPUT
      Output : Bool;
   END_VAR
   VAR_TEMP
      nTmpClock : UInt;
   END_VAR
BEGIN

REGION Network 1: Giới hạn input: Tối đa 1 phút
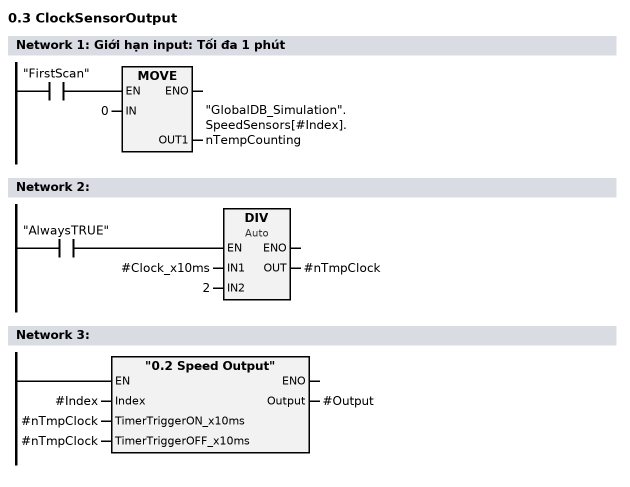
   RUNG wire#powerrail
      Contact( "FirstScan" )
      Move(in := 0, out1 => "GlobalDB_Simulation".SpeedSensors[#Index].nTempCounting)
   END_RUNG
   // the same network as SCL:
   IF "FirstScan" THEN "GlobalDB_Simulation".SpeedSensors[#Index].nTempCounting := 0; END_IF;
END_REGION

REGION Network 2
   RUNG wire#powerrail
      Contact( "AlwaysTRUE" )
      Div(in1 := #Clock_x10ms, in2 := 2, out => #nTmpClock)
   END_RUNG
   // the same network as SCL:
   IF "AlwaysTRUE" THEN #nTmpClock := #Clock_x10ms / 2; END_IF;
END_REGION

REGION Network 3
   RUNG wire#powerrail
      "0.2 Speed Output"(Index := #Index, TimerTriggerON_x10ms := #nTmpClock, TimerTriggerOFF_x10ms := #nTmpClock, Output => #Output)
   END_RUNG
   // the same network as SCL:
   "0.2 Speed Output"(Index := #Index,
                      TimerTriggerON_x10ms := #nTmpClock,
                      TimerTriggerOFF_x10ms := #nTmpClock,
                      Output => #Output);
END_REGION
END_FUNCTION

FUNCTION "0.2 Speed Output" : Void   // FC16, LAD
{ S7_Optimized_Access := 'TRUE' }
VERSION : 0.1
   VAR_INPUT
      Index : Int;
      TimerTriggerON_x10ms : UInt;   // Timebase 10ms
      TimerTriggerOFF_x10ms : UInt;   // Timebase 10ms
   END_VAR
   VAR_OUTPUT
      Output : Bool;
   END_VAR
   VAR_TEMP
      total_time : UInt;
   END_VAR
BEGIN

REGION Network 1: Giới hạn input: Tối đa 1 phút
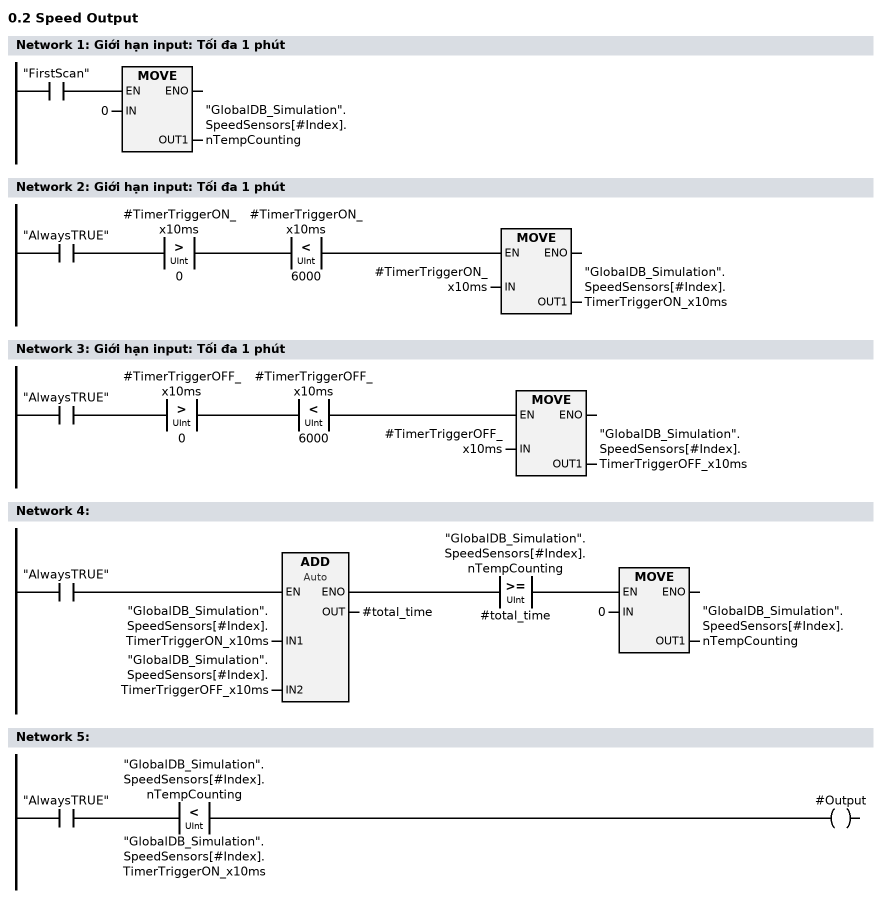
   RUNG wire#powerrail
      Contact( "FirstScan" )
      Move(in := 0, out1 => "GlobalDB_Simulation".SpeedSensors[#Index].nTempCounting)
   END_RUNG
   // the same network as SCL:
   IF "FirstScan" THEN "GlobalDB_Simulation".SpeedSensors[#Index].nTempCounting := 0; END_IF;
END_REGION

REGION Network 2: Giới hạn input: Tối đa 1 phút
   RUNG wire#powerrail
      Contact( "AlwaysTRUE" )
      { S7_Templates := "SrcType := UInt" } GT_Contact(in1 := #TimerTriggerON_x10ms, in2 := 0)
      { S7_Templates := "SrcType := UInt" } LT_Contact(in1 := #TimerTriggerON_x10ms, in2 := 6000)
      Move(in := #TimerTriggerON_x10ms, out1 => "GlobalDB_Simulation".SpeedSensors[#Index].TimerTriggerON_x10ms)
   END_RUNG
   // the same network as SCL:
   IF "AlwaysTRUE" AND (#TimerTriggerON_x10ms > 0) AND (#TimerTriggerON_x10ms < 6000) THEN
       "GlobalDB_Simulation".SpeedSensors[#Index].TimerTriggerON_x10ms := #TimerTriggerON_x10ms;
   END_IF;
END_REGION

REGION Network 3: Giới hạn input: Tối đa 1 phút
   RUNG wire#powerrail
      Contact( "AlwaysTRUE" )
      { S7_Templates := "SrcType := UInt" } GT_Contact(in1 := #TimerTriggerOFF_x10ms, in2 := 0)
      { S7_Templates := "SrcType := UInt" } LT_Contact(in1 := #TimerTriggerOFF_x10ms, in2 := 6000)
      Move(in := #TimerTriggerOFF_x10ms, out1 => "GlobalDB_Simulation".SpeedSensors[#Index].TimerTriggerOFF_x10ms)
   END_RUNG
   // the same network as SCL:
   IF "AlwaysTRUE" AND (#TimerTriggerOFF_x10ms > 0) AND (#TimerTriggerOFF_x10ms < 6000) THEN
       "GlobalDB_Simulation".SpeedSensors[#Index].TimerTriggerOFF_x10ms := #TimerTriggerOFF_x10ms;
   END_IF;
END_REGION

REGION Network 4
   RUNG wire#powerrail
      Contact( "AlwaysTRUE" )
      Add(in1 := "GlobalDB_Simulation".SpeedSensors[#Index].TimerTriggerON_x10ms, in2 := "GlobalDB_Simulation".SpeedSensors[#Index].TimerTriggerOFF_x10ms, out => #total_time)
      { S7_Templates := "SrcType := UInt" } GE_Contact(in1 := "GlobalDB_Simulation".SpeedSensors[#Index].nTempCounting, in2 := #total_time)
      Move(in := 0, out1 => "GlobalDB_Simulation".SpeedSensors[#Index].nTempCounting)
   END_RUNG
   // the same network as SCL:
   IF "AlwaysTRUE" THEN
       #total_time := "GlobalDB_Simulation".SpeedSensors[#Index].TimerTriggerON_x10ms + "GlobalDB_Simulation".SpeedSensors[#Index].TimerTriggerOFF_x10ms;
   END_IF;
   IF "AlwaysTRUE" AND ("GlobalDB_Simulation".SpeedSensors[#Index].nTempCounting >= #total_time) THEN
       "GlobalDB_Simulation".SpeedSensors[#Index].nTempCounting := 0;
   END_IF;
END_REGION

REGION Network 5
   RUNG wire#powerrail
      Contact( "AlwaysTRUE" )
      { S7_Templates := "SrcType := UInt" } LT_Contact(in1 := "GlobalDB_Simulation".SpeedSensors[#Index].nTempCounting, in2 := "GlobalDB_Simulation".SpeedSensors[#Index].TimerTriggerON_x10ms)
      Coil( #Output )
   END_RUNG
   // the same network as SCL:
   #Output := "AlwaysTRUE" AND ("GlobalDB_Simulation".SpeedSensors[#Index].nTempCounting < "GlobalDB_Simulation".SpeedSensors[#Index].TimerTriggerON_x10ms);
END_REGION
END_FUNCTION

// folder: SparePart

FUNCTION "CheckShowDataSparePart" : Void   // FC53, SCL
{ S7_Optimized_Access := 'TRUE' }
VERSION : 0.1
   VAR_INPUT
      PageMaxHMI : UDInt;
      PageCurrentHMI : UDInt;
      PageCurrentRequestServer : UDInt;
   END_VAR
   VAR_IN_OUT
      Action : Bool;
   END_VAR
   VAR_TEMP
      index_buffer : UDInt;
      index_for : UDInt;
      page_current_server : UDInt;
   END_VAR
BEGIN
   IF #Action = TRUE THEN
       IF #PageCurrentHMI >= 1 AND #PageCurrentRequestServer >= 1 AND #PageMaxHMI >= 1 THEN

           //Tính giá trị Page Server để so sánh
           #page_current_server := DINT_TO_UDINT(CEIL(UDINT_TO_REAL(#PageCurrentHMI) / 6));

           IF #page_current_server <> "DB_Machine".PageCurrentServerSparePartPrevious THEN
               "DB_Server".PageDataSparePart.PageCurrent := #page_current_server;
               "DB_Server".ActionSearchLossSparePart := 1;

               "DB_Machine".PageCurrentServerSparePartPrevious := #page_current_server;
           ELSE
               IF "DB_Server".ActionSearchLossSparePart = 2 OR "DB_Server".ActionSearchLossSparePart = 3 THEN
                   // //Check xem có data sẵn chưa
                   // IF #PageCurrentHMI <= #PageMaxHMI THEN
                   //     #index_buffer := #PageCurrentHMI MOD 6;
                   //     IF #index_buffer = 0 THEN
                   //         #index_buffer := 6;
                   //     END_IF;

                   //     #index_buffer := (#index_buffer - 1) * 5;

                   //     FOR #index_for := 1 TO 5 DO
                   //         "DB_DataHMI".DataSparePartShowHmiDTO[#index_for]."No." := (#PageCurrentHMI - 1) * 5 + #index_for;
                   //         "DB_DataHMI".DataSparePartShowHmiDTO[#index_for].Name := "BufferServerSend".buffer_spare_part[#index_buffer + #index_for].name;
                   //         "DB_DataHMI".DataSparePartShowHmiDTO[#index_for].ProductCount := "BufferServerSend".buffer_spare_part[#index_buffer + #index_for].product_count;

                   //         "DTL_to_StringV2"("DTL" := "BufferServerSend".buffer_spare_part[#index_buffer + #index_for].start_time,
                   //                           DateTimeString => "DB_DataHMI".DataSparePartShowHmiDTO[#index_for].StartTime);

                   //         "DTL_to_StringV2"("DTL" := "BufferServerSend".buffer_spare_part[#index_buffer + #index_for].end_time,
                   //                           DateTimeString => "DB_DataHMI".DataSparePartShowHmiDTO[#index_for].EndTime);

                   //         IF "BufferServerSend".buffer_spare_part[#index_buffer + #index_for].name='' THEN
                   //             "DB_DataHMI".DataSparePartShowHmiDTO[#index_for].IsHaveData := FALSE;
                   //         ELSE
                   //             "DB_DataHMI".DataSparePartShowHmiDTO[#index_for].IsHaveData := TRUE;
                   //         END_IF;

                   //     END_FOR;
                   // END_IF;
                   #Action := FALSE;
               END_IF;
           END_IF;
       END_IF;
   END_IF;

   // // //Check xem có data sẵn chưa
   IF #PageCurrentHMI <= #PageMaxHMI THEN
       #index_buffer := #PageCurrentHMI MOD 6;
       IF #index_buffer = 0 THEN
           #index_buffer := 6;
       END_IF;

       #index_buffer := (#index_buffer - 1) * 5;

       FOR #index_for := 1 TO 5 DO
           "DB_DataHMI".DataSparePartShowHmiDTO[#index_for]."No." := (#PageCurrentHMI - 1) * 5 + #index_for;
           "DB_DataHMI".DataSparePartShowHmiDTO[#index_for].Name := "BufferServerSend".buffer_spare_part[#index_buffer + #index_for].name;
           "DB_DataHMI".DataSparePartShowHmiDTO[#index_for].ProductCount := "BufferServerSend".buffer_spare_part[#index_buffer + #index_for].product_count;

           "DTL_to_StringV2"("DTL" := "BufferServerSend".buffer_spare_part[#index_buffer + #index_for].start_time,
                             DateTimeString => "DB_DataHMI".DataSparePartShowHmiDTO[#index_for].StartTime);

           "DTL_to_StringV2"("DTL" := "BufferServerSend".buffer_spare_part[#index_buffer + #index_for].end_time,
                             DateTimeString => "DB_DataHMI".DataSparePartShowHmiDTO[#index_for].EndTime);

           IF "BufferServerSend".buffer_spare_part[#index_buffer + #index_for].name = '' THEN
               "DB_DataHMI".DataSparePartShowHmiDTO[#index_for].IsHaveData := FALSE;
           ELSE
               "DB_DataHMI".DataSparePartShowHmiDTO[#index_for].IsHaveData := TRUE;
           END_IF;

       END_FOR;
   END_IF;
END_FUNCTION

// ===== PLC "MqttPlc1500"  CPU 1517F-3 PN/DP =====

// folder: Common

TYPE "typeDiagnostics"
TITLE = typeDiagnostics
// Provides a structure for detailed diagnostics
   STRUCT
      status : Word;   // Status of the block or error identification when error occurred
      subfunctionStatus : DWord;   // Status or return value of called FBs, FCs and system blocks
      stateNumber : DInt;   // State in the state machine of the block where the error occurred
   END_STRUCT;
END_TYPE

// folder: LMQTT

TYPE "LMQTT_typeConnParam"
TITLE = LMQTT_typeConnParams
// Specifies connection parameters for the mqtt connection
   STRUCT
      hwId : Hw_Any;   // Hardware identifier of the interface. 0: interface is selected automatically
      connId : Conn_Ouc := 1;   // Unique connection identifier (1..4095)
      broker : String;   // Hostname or IP address of broker
      port : UInt := 1883;   // Port on the broker
      tls : Struct   // Parameters for TLS encryption
         enableTls : Bool;   // TRUE: Enables TLS, FALSE: disable TLS
         validateServerIdentity : Bool;   // TRUE: Validate server certificate, FALSE: No validation of server certificate
         brokerCert : UDInt;   // ID of the broker's certificate in TIA Portal
         clientCert : UDInt;   // ID of the client's certificate in TIA Portal
      END_STRUCT;
      keepAlive : UInt;   // Keepalive mechanism for MQTT in seconds. 0: disabled.
   END_STRUCT;
END_TYPE

// folder: (top level)

DATA_BLOCK "InstLMQTT_Client"   // DB1
{ S7_Optimized_Access := 'TRUE' }
AUTHOR : SiemensAG
FAMILY : MQTT
VERSION : 1.0
// stored: InstanceOfName LMQTT_Client
"LMQTT_Client"
BEGIN
END_DATA_BLOCK

DATA_BLOCK "MqttDb"   // DB2
TITLE = Configuration Data block example for LMQTT_Client
{ S7_Optimized_Access := 'TRUE' }
AUTHOR : Siemens
FAMILY : LMQTT
VERSION : 1.0
// This block is an example how to control the LMQTT_Client function block
   VAR
      control : Struct   // Input of the FB
         enable : Bool;   // Set TRUE, to establish a connection - set to FALSE to disconnect
         publish : Bool;   // Rising Edge: Sends a message
         subscribe : Bool;   // Rising Edge: Subscribes to a topic
         unsubscribe : Bool;   // Rising Edge: Unsubscribes to a topic
      END_STRUCT;
      output : Struct   // Output Information of the FB
         valid : Bool;   // TRUE: Valid set of output values available at the FB
         done : Bool;   // TRUE: If last Request was successfull
         busy : Bool;   // TRUE: FB is not finished and new output values can be expected
         error : Bool;   // TRUE: An error occurred during the execution of the FB
         status : Word;   // 16#0000 - 16#7FFF: Status of the FB, 16#8000 - 16#FFFF: Error identification
         diagnostics : "typeDiagnostics";   // Diagnostics information of FB (optional)
      END_STRUCT;
      connParam : "LMQTT_typeConnParam";   // Connection Parameters
      clientIdentifier : WString[20];   // ClientId with one or more characters
      username : WString[20];   // Username used for connect
      password : WString[20];   // Password used for connect
      willTopic : WString[20];   // Topic where the last will message is sent
      willMsgPayload : Array[0..99] of Byte;   // Last will message Data - valid bytes in this array must be written in input 'willMsgLen'
      willMsgLen : UInt;   // Valid number of elements in Will Message Data Array. Max 65535 Byte allowed by MQTT Spec.
      qos : USInt;   // Sets QoS 0,1 or 2 for the Publish and Will Message - Subscribe only allows QoS 0 and 1
      mqttTopic : WString[100];   // Mqtt Topic to Publish / Subscribe / Unsubscribe
      publishMsgPayload : Array[0..999] of Byte;   // Message Data to Publish - valid bytes in this array must be written in input 'publishMsgLen'
      publishMsgLen : UDInt;   // Valid number of elements in publish message data Array
      retain : Bool;   // TRUE: Published Message will be set to retain on MQTT broker
      receivedTopic : WString[200];   // Mqtt Topic of received message
      receivedMsgPayload : Array[0..999] of Byte;   // Mqtt message data that was received - valid bytes in this array indicated by 'receivedMsgDataLen' output
      receivedMsgDataLen : UDInt;   // Amount of Bytes received in receivedMessage INOUT area
      receivedMsgStatus : USInt;   // 0: No new Message, 1: New valid Message received and available at InOut area, 2: New message, but data is invalid (wrong message len or message could not be copied to InOut received topic or received message)
   END_VAR
BEGIN
   willMsgPayload[0] := 16#6F;
   willMsgPayload[1] := 16#66;
   willMsgPayload[2] := 16#66;
   willMsgPayload[3] := 16#6C;
   willMsgPayload[4] := 16#69;
   willMsgPayload[5] := 16#6E;
   willMsgPayload[6] := 16#65;
   publishMsgPayload[1] := 16#65;
   publishMsgPayload[2] := 16#6c;
   publishMsgPayload[3] := 16#6c;
   publishMsgPayload[4] := 16#6f;
   publishMsgPayload[5] := 16#20;
   publishMsgPayload[6] := 16#77;
   publishMsgPayload[7] := 16#6f;
   publishMsgPayload[8] := 16#72;
   publishMsgPayload[9] := 16#6c;
   publishMsgPayload[10] := 16#64;
   publishMsgPayload[0] := 16#68;
END_DATA_BLOCK

ORGANIZATION_BLOCK "Main"   // OB1, LAD, ProgramCycle
TITLE = "Main Program Sweep (Cycle)"
{ S7_Optimized_Access := 'TRUE' }
VERSION : 0.1
   VAR_INPUT
      Initial_Call : Bool;   // Initial call of this OB
      Remanence : Bool;   // =True, if remanent data are available
   END_VAR
   VAR_TEMP
      tempC : DInt;
   END_VAR
BEGIN

REGION Network 1
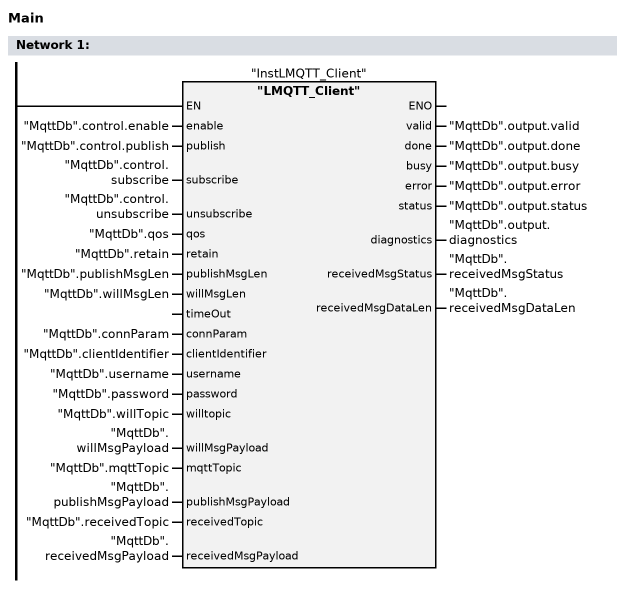
   RUNG wire#powerrail
      "InstLMQTT_Client"(enable := "MqttDb".control.enable, publish := "MqttDb".control.publish, subscribe := "MqttDb".control.subscribe, unsubscribe := "MqttDb".control.unsubscribe, qos := "MqttDb".qos, retain := "MqttDb".retain, publishMsgLen := "MqttDb".publishMsgLen, willMsgLen := "MqttDb".willMsgLen, timeOut :=, connParam := "MqttDb".connParam, clientIdentifier := "MqttDb".clientIdentifier, username := "MqttDb".username, password := "MqttDb".password, willtopic := "MqttDb".willTopic, willMsgPayload := "MqttDb".willMsgPayload, mqttTopic := "MqttDb".mqttTopic, publishMsgPayload := "MqttDb".publishMsgPayload, receivedTopic := "MqttDb".receivedTopic, receivedMsgPayload := "MqttDb".receivedMsgPayload, valid => "MqttDb".output.valid, done => "MqttDb".output.done, busy => "MqttDb".output.busy, error => "MqttDb".output.error, status => "MqttDb".output.status, diagnostics => "MqttDb".output.diagnostics, receivedMsgStatus => "MqttDb".receivedMsgStatus, receivedMsgDataLen => "MqttDb".receivedMsgDataLen)
   END_RUNG
   // the same network as SCL:
   "InstLMQTT_Client"(enable := "MqttDb".control.enable,   // "LMQTT_Client"
                      publish := "MqttDb".control.publish,
                      subscribe := "MqttDb".control.subscribe,
                      unsubscribe := "MqttDb".control.unsubscribe,
                      qos := "MqttDb".qos,
                      retain := "MqttDb".retain,
                      publishMsgLen := "MqttDb".publishMsgLen,
                      willMsgLen := "MqttDb".willMsgLen,
                      connParam := "MqttDb".connParam,
                      clientIdentifier := "MqttDb".clientIdentifier,
                      username := "MqttDb".username,
                      password := "MqttDb".password,
                      willtopic := "MqttDb".willTopic,
                      willMsgPayload := "MqttDb".willMsgPayload,
                      mqttTopic := "MqttDb".mqttTopic,
                      publishMsgPayload := "MqttDb".publishMsgPayload,
                      receivedTopic := "MqttDb".receivedTopic,
                      receivedMsgPayload := "MqttDb".receivedMsgPayload,
                      valid => "MqttDb".output.valid,
                      done => "MqttDb".output.done,
                      busy => "MqttDb".output.busy,
                      error => "MqttDb".output.error,
                      status => "MqttDb".output.status,
                      diagnostics => "MqttDb".output.diagnostics,
                      receivedMsgStatus => "MqttDb".receivedMsgStatus,
                      receivedMsgDataLen => "MqttDb".receivedMsgDataLen);
END_REGION
END_ORGANIZATION_BLOCK

// folder: Common

FUNCTION "IsIPAddress" : Bool   // FC1, SCL
TITLE = IsIPAddress
{ S7_Optimized_Access := 'TRUE' }
VERSION : 0.1
// Evaluates whether a given String contains a valid IP address
   VAR_INPUT
      address : String;   // Address to be evaluated
   END_VAR
   VAR_OUTPUT
      ipAddress : IP_V4;   // Parsed IP address if passed address is IP address
   END_VAR
   VAR_TEMP
      tempAddress : String;   // Passed address
      tempOctet : String;   // Current octet
      tempIndex : DInt;   // Index for loop
      tempPos : Int;   // Position of found separator
      tempNum : Int;   // Converted octet
      tempIp : IP_V4;   // Parsed IP address
   END_VAR
   // Ret_Val : Return value
   VAR CONSTANT
      MAX_VALUE : USInt := 255;   // Max. valid value of octet
      NUM_OCTETS : DInt := 4;   // Number of octets
      CHAR_ZERO : Char := '0';   // ASCII character '0'
   END_VAR
BEGIN
   REGION BLOCK INFO HEADER
     //===============================================================================
     // SIEMENS / (c)Copyright 2024
     //-------------------------------------------------------------------------------
     // Title:        IsIPAddress
     // Function:     Evaluates whether a given String contains a valid IP address
     // Library:      --
     // Author:       Siemens Industry Online Support
     // Tested with:  CPU 1515-2 PN V3.1
     // Engineering:  TIA Portal V17
     // Restrictions: --
     // Requirements: S7-1200 with firmware V4.4 or higher
     //               S7-1500 with firmware V2.0 or higher
     //-------------------------------------------------------------------------------
     // Change log table:
     // Version  | Date       | Expert in charge       | Changes applied
     //-------------------------------------------------------------------------------
     // 01.00.00 | 2024-02-12 | Online Support         | First released version
     //===============================================================================
   END_REGION

   #tempAddress := #address;
   #IsIPAddress := FALSE; // Will be overwritten if IP address is detected
   #ipAddress := #tempIp; // Zero output parameter

   FOR #tempIndex := 1 TO #NUM_OCTETS DO
     #tempPos := FIND(IN1 := #tempAddress, IN2 := '.'); // Find separator

     IF (#tempPos > 0 OR #tempIndex = #NUM_OCTETS) // Separator found with exception of last octet
       AND NOT (#tempPos > 0 AND #tempIndex = #NUM_OCTETS) // No separator found in last octet
       AND #tempPos <= 4 // 3  characters or less
     THEN
       IF #tempIndex < #NUM_OCTETS THEN // First three octets
         #tempOctet := LEFT(IN := #tempAddress, L := #tempPos - 1);
       ELSE// Last octet
         #tempOctet := #tempAddress;
       END_IF;

       STRG_VAL(IN := #tempOctet,
                FORMAT := 0,
                P := 1,
                OUT => #tempNum);

       IF #tempNum >= 0 AND #tempNum <= #MAX_VALUE // Within 0 and 255
         AND NOT (#tempNum = 0 AND #tempIndex = 1) // Not 0 in first octet
         AND NOT (#tempNum = 0 AND #tempOctet[1] <> #CHAR_ZERO) // Not 0 because of invalid character
       THEN
         #tempIp.ADDR[#tempIndex] := INT_TO_BYTE(#tempNum);
         #tempAddress := RIGHT(IN := #tempAddress, L := LEN(#tempAddress) - #tempPos); // Remove evaluated octet
       ELSE // Address is not IP address
         EXIT;
       END_IF;
     ELSE // Address is not IP address
       EXIT;
     END_IF;

     IF #tempIndex = #NUM_OCTETS THEN // End of loop reached, address is IP address
       #ipAddress := #tempIp;
       #IsIPAddress := true;
     END_IF;
   END_FOR;
END_FUNCTION

// folder: LMQTT

